// SIMATIC STEP 7 (V5.x) project R706_Cogeme_V_0_2
// CPU: CPU 315-2 DP
// station: Hardware
// station: R706_Ass_3PCS_Insert
// station: P_ADR_BUS
// program: Programma S7(1)
// program: Backup  DB 20100406
// program: SINAMICS_S120_CU310_DP
// program: SINAMICS_S120_CU310_DP

SYMBOL_TABLE
"Line"	DB 50	UDT 250
"Line.MapE"	DB 51	DB 51
"Line.MapA"	DB 52	DB 52
"Line.Config"	DB 53	DB 53
"Line.Alarms"	DB 54	DB 54
"Line.Systems"	DB 55	DB 55
"Line.Cycles"	DB 60	DB 60
"Line.OperatorPanel"	DB 70	DB 70
"OP10"	DB 100	UDT 250
"Op10.Bench.MapE"	DB 101	DB 101
"Op10.Bench.MapA"	DB 102	DB 102
"Op10.Bench.Config"	DB 103	DB 103
"Op10.Bench.Alarms"	DB 104	DB 104
"Op10.Bench.Systems"	DB 105	DB 105
"Op10.Tools.MapE"	DB 106	DB 106
"Op10.Tools.Config"	DB 108	DB 108
"Op10.Tools.Systems"	DB 109	DB 109
"Op10.Bench.Recipe"	DB 110	DB 110
"Op10.Cycles"	DB 120	DB 120
"OP20"	DB 150	UDT 250
"Op20.Bench.MapE"	DB 151	DB 151
"Op20.Bench.MapA"	DB 152	DB 152
"Op20.Bench.Config"	DB 153	DB 153
"Op20.Bench.Alarms"	DB 154	DB 154
"Op20.Bench.Systems"	DB 155	DB 155
"Op20.Tools.MapE"	DB 156	DB 156
"Op20.Tools.Config"	DB 158	DB 158
"Op20.Tools.Systems"	DB 159	DB 159
"Op20.Bench.Recipe"	DB 160	DB 160
"Op20.Cycles"	DB 170	DB 170
"OP40"	DB 200	UDT 250
"Op40.Bench.MapE"	DB 201	DB 201
"Op40.Bench.MapA"	DB 202	DB 202
"Op40.Bench.Config"	DB 203	DB 203
"Op40.Bench.Alarms"	DB 204	DB 204
"Op40.Bench.Systems"	DB 205	DB 205
"Op40.Tools.MapE"	DB 206	DB 206
"Op40.Tools.Config"	DB 208	DB 208
"Op40.Tools.Systems"	DB 209	DB 209
"Op40.Bench.Recipe"	DB 210	DB 210
"Op40.Cycles"	DB 220	DB 220
"Op05.Bench"	DB 300	UDT 250
"Ist_cil_10_Index_cass"	DB 401	FB 102
"Ist_10_CilBloccoPezzo"	DB 402	FB 102
"Ist_cil_20_Index_cass"	DB 403	FB 102
"Ist_cil_20_gr_piantaggio"	DB 404	FB 102
"Ist_cil_20_piantaggio"	DB 405	FB 102
"Ist_cil_40_Index_cass"	DB 406	FB 102
"Ist_40_CilBloccoPezzo"	DB 407	FB 102
"Ist_AsseX"	DB 420	FB 450
"Ist_AsseY"	DB 421	FB 450
"Ist_CU_asseX"	DB 425	FB 455
"Ist_CU_asseY"	DB 426	FB 455
"Op10.Ist.Cycle.General"	DB 430	FB 120
"Op10.Ist.Cycle.Restore"	DB 431	FB 121
"OP40.Ist.Cycle.Restore"	DB 435	FB 221
"OP40.Ist.Cycle.General"	DB 436	FB 220
"OP20.Ist.Cycle.Restore"	DB 437	FB 171
"OP20.Ist.Cycle.General"	DB 438	FB 170
"Line.Ist.Cycle.Coord_rib"	DB 440	FB 60
"Line.Cycle.Coord_ribadit"	FB 60	FB 60	// Coordinamento ribaditrice
"Std System.Cylinder"	FB 102	FB 102
"Op10.Cycle.General"	FB 120	FB 120
"Op10.Cycle.Restore"	FB 121	FB 121
"Op20.Cycle.General"	FB 170	FB 170
"Op20.Cycle.Restore"	FB 171	FB 171
"Op40.Cycle.General"	FB 220	FB 220
"Op40.Cycle.Restore"	FB 221	FB 221
"Std_Sinamics_Axis"	FB 450	FB 450
"Std.Sinamics_Cu_S"	FB 455	FB 455
"SCALE"	FC 5	FC 5	// Scaling Values
"Conv_INT->BIT"	FC 17	FC 17
"Bench.Mode"	FC 20	FC 20
"Bench.Alarms"	FC 21	FC 21	// Da ricontrollare!!!!
"TIM_S5TI"	FC 40	FC 40	// IEC Time to S5 Time
"Line.FCMain"	FC 50	FC 50
"Line.FCMapE"	FC 51	FC 51
"Line.FCMapA"	FC 52	FC 52
"Line.FCConfig"	FC 53	FC 53
"Line.FCSystems"	FC 55	FC 55
"Line.FCCycles"	FC 60	FC 60
"Line.FCOperatorPanel"	FC 70	FC 70
"OP10.FCMain"	FC 100	FC 100
"Op10.Bench.FCMapE"	FC 101	FC 101
"Op10.Bench.FCMapA"	FC 102	FC 102
"Op10.Bench.FCConfig"	FC 103	FC 103
"Op10.Bench.FCSystems"	FC 105	FC 105
"Op10.Tool.FCMap.E"	FC 106	FC 106
"Op10.FCCycles"	FC 120	FC 120
"OP20.FCMain"	FC 150	FC 150
"Op20.Bench.FCMapE"	FC 151	FC 151
"Op20.Bench.FCMapA"	FC 152	FC 152
"Op20.Bench.FCConfig"	FC 153	FC 153
"Op20.Bench.FCSystems"	FC 155	FC 155
"Op20.Tool.FCMapE"	FC 156	FC 156
"Op20.FCCycles"	FC 170	FC 170
"OP40.FCMain"	FC 200	FC 200
"Op40.Bench.FCMapE"	FC 201	FC 201
"Op40.Bench.FCMapA"	FC 202	FC 202
"Op40.Bench.FCConfig"	FC 203	FC 203
"Op40.Bench.FCSystems"	FC 205	FC 205
"Op40.Tool.FCMapE"	FC 206	FC 206
"Op40.FCCycles"	FC 220	FC 220
"Dummy_ReferenceAxX"	M 10.0	BOOL
"Dummy_RefCamAxX"	M 10.1	BOOL
"Dummy_ReferenceAxY"	M 10.2	BOOL
"Dummy_RefCamAxY"	M 10.3	BOOL
"AppoFP_M50.0"	M 50.0	BOOL
"AppoFP_M50.1"	M 50.1	BOOL
"AppoFP_M50.2"	M 50.2	BOOL
"AppoFP_M50.3"	M 50.3	BOOL
"AppoFP_M50.4"	M 50.4	BOOL
"AppoFP_M50.5"	M 50.5	BOOL
"AppoFP_M50.6"	M 50.6	BOOL
"AppoFP_M50.7"	M 50.7	BOOL
"AppoFP_M51.0"	M 51.0	BOOL
"AppoFP_M51.1"	M 51.1	BOOL
"AppoFPM51.2"	M 51.2	BOOL
"AppoFPM51.3"	M 51.3	BOOL
"AppoFPM51.4"	M 51.4	BOOL
"AppoFPM51.5"	M 51.5	BOOL
"AppoFP_M51.6"	M 51.6	BOOL
"AppoFP_M51.7"	M 51.7	BOOL
"AppoFP_M52.0"	M 52.0	BOOL
"Alw_ON"	M 100.0	BOOL
"alw_OFF"	M 100.1	BOOL
"FirstScan"	M 100.2	BOOL
"M100.3"	M 100.3	BOOL
"FP_manual"	M 100.4	BOOL
"M100.5"	M 100.5	BOOL
"Fp_Automatic"	M 100.6	BOOL
"Clock-T=0,1 sec."	M 250.0	BOOL
"Clock-T=0,2 sec."	M 250.1	BOOL
"Clock-T=0,4 sec."	M 250.2	BOOL
"Clock-T=0,5 sec."	M 250.3	BOOL
"Clock-T=0,8 sec."	M 250.4	BOOL
"Clock-T=1 sec."	M 250.5	BOOL
"Clock-T=1,6 sec."	M 250.6	BOOL
"Clock-T=2 sec."	M 250.7	BOOL
"I/O_FLT1"	OB 82	OB 82	// I/O Point Fault 1
"RACK_FLT"	OB 86	OB 86	// Loss of Rack Fault
"TON"	SFB 4	SFB 4	// Generate an On Delay
"DPRD_DAT"	SFC 14	SFC 14	// Read Consistent Data of a Standard DP Slave
"DPWR_DAT"	SFC 15	SFC 15	// Write Consistent Data to a Standard DP Slave
"TempoResetAllarmi"	T 2	TIMER
"T_All_Rientro_PLC_OK"	T 3	TIMER
"T_Allarme_aria_compressa"	T 5	TIMER
"Rit_all_potre_non_blocc"	T 6	TIMER
"Op10_Tempo_di_ribaditura"	T 10	TIMER
"Op40_Tempo_di_ribaditura"	T 11	TIMER
"TOP20_Cassetto dentro"	T 20	TIMER
"OP20_TimeoutPiantaggio"	T 21	TIMER
"OP20_TempoDiPiantaggio"	T 22	TIMER
"OP10St13_Cassetto_dentro"	T 25	TIMER
"OP10St35_Cassetto_fuori"	T 26	TIMER
"RP10St15_Cassetto_fuori"	T 27	TIMER
"OP20ST10_Cassetto_dentro"	T 28	TIMER
"OP40St13_Cassetto_dentro"	T 29	TIMER
"OP40St35_Cassetto_fuori"	T 30	TIMER
"RS40St15_Cassetto_fuori"	T 31	TIMER
"Cycles_UDT"	UDT 200	UDT 200
"Bench_UDT"	UDT 250	UDT 250
"Sinamics Telegramma Assi"	UDT 450	UDT 450
"Sinamics TelegrammaCU_S"	UDT 455	UDT 455
"Assi e posizioni"	VAT 1	
END_SYMBOL_TABLE

TYPE "Cycles_UDT"	// UDT 200
VERSION : 0.1
  STRUCT
   State : STRUCT
    State : INT ;	//Stato del ciclo
    Page : INT ;	//Pagina
    Message : INT ;	//Messaggio
    Cycle_In_Progress : BOOL ;	//Ciclo in corso
    Cycle_Ended_OK : BOOL ;	//Ciclo terminato OK
    Cycle_Ended_KO : BOOL ;	//Ciclo terminato KO
    State_Bit : ARRAY  [0 .. 63 ] OF //Bit Stato
    BOOL ;
    Free : INT ;
   END_STRUCT ;
   Command : STRUCT
    Activate_Cycle : BOOL ;	//Attiva ciclo
    Hold_Cycle : BOOL ;	//Sospendi ciclo
    Single_Step : BOOL ;	//Passo singolo
    Lock_Outputs : BOOL ;	//Blocco uscite
    Free : INT ;
   END_STRUCT ;
  END_STRUCT ;	
END_TYPE

TYPE "Bench_UDT"	// UDT 250
VERSION : 0.1
  STRUCT
   Mode : STRUCT
    Emergency : BOOL ;	//MODO Macchina spenta
    Test_Machine : BOOL ;	//MODO Aspetta pressione nel circuito pneumatico e/o idraulico + MODO Test Lampad
    Setup : BOOL ;	//MODO Cambio Ricetta o setup
    Manual : BOOL ;	//MODO Manuale
    Automatic : BOOL ;	//MODO Automatico
    Service : BOOL ;	//MODO Messa in servizio
    Free_06 : BOOL ;
    Free_07 : BOOL ;
   END_STRUCT ;
   Diagnostic : STRUCT
    Alarm_Emergency : BOOL ;	//Macchina in Emergenza
    Alarm_Stop_Cycle : BOOL ;	//Allarme che blocca il ciclo attivo
    Alarm_No_Restart : BOOL ;	//Allarme che blocca un nuovo ciclo
    Alarm_Warning : BOOL ;	//Segnalazione o avvertenza
    Safe_State : BOOL ;	//MODO Sicuro : e' possibile eseguire i comandi manuali in sicurezza
    Initial_Conditions : BOOL ;	//condizioni iniziali macchina
    Hold_State : BOOL ;	//Hold Macchina
    Free_07 : BOOL ;
    ResetAlarm : BOOL ;
   END_STRUCT ;
   Software : STRUCT
    SwName : STRING  [20 ];
    SwVersion : STRING  [11 ];
   END_STRUCT ;
  END_STRUCT ;	
END_TYPE

TYPE "Sinamics Telegramma Assi"	// UDT 450
AUTHOR : Castel
VERSION : 0.1
  STRUCT
   IN : STRUCT
    IN_PZD1_BIT8 : BOOL ;	//PAST1 Bit8 distanza di inseguimento nella tolleranza (1=si 0=no)
    IN_PZD1_BIT9 : BOOL ;	//PAST1 Bit9 comando richiesto (1=si 0=no)
    IN_PZD1_BIT10 : BOOL ;	//PAST1 Bit10 posizione di destinazione raggiunta (1=si 0=no)
    IN_PZD1_BIT11 : BOOL ;	//PAST1 Bit11 punto di riferimento impostato (1=si 0=no)
    IN_PZD1_BIT12 : BOOL ;	//PAST1 Bit12 tacitazione blocco movimento attivata (1=si 0=no)
    IN_PZD1_BIT13 : BOOL ;	//PAST1 Bit13 (motore fermo) n_att< valore di soglia num.giri 3 P2161 (1=si 0=no)
    IN_PZD1_BIT14 : BOOL ;	//PAST1 Bit14 riservato
    IN_PZD1_BIT15 : BOOL ;	//PAST1 Bit15 riservato
    IN_PZD1_BIT0 : BOOL ;	//PAST1 Bit0 pronto all'inserzione (1=si 0=no)
    IN_PZD1_BIT1 : BOOL ;	//PAST1 Bit1 pronto al funzionamento (1=si 0=no)
    IN_PZD1_BIT2 : BOOL ;	//PAST1 Bit2 funzionamento abilitazione (1=si 0=no)
    IN_PZD1_BIT3 : BOOL ;	//PAST1 Bit3 anomalia attiva (1=si 0=no)
    IN_PZD1_BIT4 : BOOL ;	//PAST1 Bit4 nessun arresto per inerzia attivo (1=OFF2 inattivo 0=OFF2 attivo)
    IN_PZD1_BIT5 : BOOL ;	//PAST1 Bit5 nessun arresto rapido attivo (1=OFF3 inattivo 0=OFF3 attivo)
    IN_PZD1_BIT6 : BOOL ;	//PAST1 Bit6 blocco inserzione attivo (1=si 0=no)
    IN_PZD1_BIT7 : BOOL ;	//PAST1 Bit7 avviso attivo (1=si 0=no)
    IN_PZD2_BIT8 : BOOL ;	//AKTSATZ Bit8
    IN_PZD2_BIT9 : BOOL ;	//AKTSATZ Bit9
    IN_PZD2_BIT10 : BOOL ;	//AKTSATZ Bit10
    IN_PZD2_BIT11 : BOOL ;	//AKTSATZ Bit11
    IN_PZD2_BIT12 : BOOL ;	//AKTSATZ Bit12
    IN_PZD2_BIT13 : BOOL ;	//AKTSATZ Bit13
    IN_PZD2_BIT14 : BOOL ;	//AKTSATZ Bit14 attivare il cambio del blocco esterno
    IN_PZD2_BIT15 : BOOL ;	//AKTSATZ Bit15 MDI attivo (1=attivo 0=inattivo)
    IN_PZD2_BIT0 : BOOL ;	//AKTSATZ Bit0 blocco di movimento attivo valenza 0 (1=attivo 0=inattivo)
    IN_PZD2_BIT1 : BOOL ;	//AKTSATZ Bit1 blocco di movimento attivo valenza 2 (1=attivo 0=inattivo)
    IN_PZD2_BIT2 : BOOL ;	//AKTSATZ Bit2 blocco di movimento attivo valenza 4 (1=attivo 0=inattivo)
    IN_PZD2_BIT3 : BOOL ;	//AKTSATZ Bit3 blocco di movimento attivo valenza 8 (1=attivo 0=inattivo)
    IN_PZD2_BIT4 : BOOL ;	//AKTSATZ Bit4 blocco di movimento attivo valenza 16 (1=attivo 0=inattivo)
    IN_PZD2_BIT5 : BOOL ;	//AKTSATZ Bit5 blocco di movimento attivo valenza 32 (1=attivo 0=inattivo)
    IN_PZD2_BIT6 : BOOL ;	//AKTSATZ Bit6
    IN_PZD2_BIT7 : BOOL ;	//AKTSATZ Bit7
    IN_PZD3_BIT8 : BOOL ;	//POSPAST Bit8 valore attuale di posiz. <= posiz.commutazione camma 1 (1=si 0=no)
    IN_PZD3_BIT9 : BOOL ;	//POSPAST Bit9 valore attuale di posiz. <= posiz.commutazione camma 2 (1=si 0=no)
    IN_PZD3_BIT10 : BOOL ;	//POSPAST Bit10 uscita diretta 1 su blocco di movimento (1=si 0=no)
    IN_PZD3_BIT11 : BOOL ;	//POSPAST Bit11 uscita diretta 2 su blocco di movimento (1=si 0=no)
    IN_PZD3_BIT12 : BOOL ;	//POSPAST Bit12
    IN_PZD3_BIT13 : BOOL ;	//POSPAST Bit13
    IN_PZD3_BIT14 : BOOL ;	//POSPAST Bit14
    IN_PZD3_BIT15 : BOOL ;	//POSPAST Bit15
    IN_PZD3_BIT0 : BOOL ;	//POSPAST Bit0 funzionamento a seguire attivo (1=si 0=no)
    IN_PZD3_BIT1 : BOOL ;	//POSPAST Bit1 limitazione di velocità attiva (1=si 0=no)
    IN_PZD3_BIT2 : BOOL ;	//POSPAST Bit2 valore di riferimento fermo (1=si 0=no)
    IN_PZD3_BIT3 : BOOL ;	//POSPAST Bit3
    IN_PZD3_BIT4 : BOOL ;	//POSPAST Bit4 asse in movimento avanti (1=si 0=no)
    IN_PZD3_BIT5 : BOOL ;	//POSPAST Bit5 asse in movimento indietro (1=si 0=no)
    IN_PZD3_BIT6 : BOOL ;	//POSPAST Bit6 finecorsa software meno raggiunto (1=si 0=no)
    IN_PZD3_BIT7 : BOOL ;	//POSPAST Bit7 finecorsa software più raggiunto (1=si 0=no)
    IN_PZD4_BIT8 : BOOL ;	//PAST2 Bit8 posizionamento su riscontro fisso attivo (1=si 0=no)
    IN_PZD4_BIT9 : BOOL ;	//PAST2 Bit9
    IN_PZD4_BIT10 : BOOL ;	//PAST2 Bit10
    IN_PZD4_BIT11 : BOOL ;	//PAST2 Bit11 commutazione record di dati motore attiva (1=attivo 0=inattivo)
    IN_PZD4_BIT12 : BOOL ;	//PAST2 Bit12 segno di vita dello slave bit 0 (1=on 0=off)
    IN_PZD4_BIT13 : BOOL ;	//PAST2 Bit13 segno di vita dello slave bit 1 (1=on 0=off)
    IN_PZD4_BIT14 : BOOL ;	//PAST2 Bit14 segno di vita dello slave bit 2 (1=on 0=off)
    IN_PZD4_BIT15 : BOOL ;	//PAST2 Bit15 segno di vita dello slave bit 3 (1=on 0=off)
    IN_PZD4_BIT0 : BOOL ;	//PAST2 Bit0 DDS attivo bit 0 (1=on 0=off)
    IN_PZD4_BIT1 : BOOL ;	//PAST2 Bit1 DDS attivo bit 1 (1=on 0=off)
    IN_PZD4_BIT2 : BOOL ;	//PAST2 Bit2 DDS attivo bit 2 (1=on 0=off)
    IN_PZD4_BIT3 : BOOL ;	//PAST2 Bit3 DDS attivo bit 3 (1=on 0=off)
    IN_PZD4_BIT4 : BOOL ;	//PAST2 Bit4 DDS attivo bit 4 (1=on 0=off)
    IN_PZD4_BIT5 : BOOL ;	//PAST2 Bit5
    IN_PZD4_BIT6 : BOOL ;	//PAST2 Bit6
    IN_PZD4_BIT7 : BOOL ;	//PAST2 Bit7 asse in sosta attivo (1=si 0=no)
    IN_PZD5_BIT8 : BOOL ;	//SEGNW Bit8 diff.val.rif./att.n.giri entro tolleranza t_on (1=si 0=no)
    IN_PZD5_BIT9 : BOOL ;	//SEGNW Bit9
    IN_PZD5_BIT10 : BOOL ;	//SEGNW Bit10
    IN_PZD5_BIT11 : BOOL ;	//SEGNW Bit11 abilitazione regolatore (1=si 0=no)
    IN_PZD5_BIT12 : BOOL ;	//SEGNW Bit12 azionamento pronto (1=si 0=no)
    IN_PZD5_BIT13 : BOOL ;	//SEGNW Bit13 impulsi abilitati (1=si 0=no)
    IN_PZD5_BIT14 : BOOL ;	//SEGNW Bit14
    IN_PZD5_BIT15 : BOOL ;	//SEGNW Bit15
    IN_PZD5_BIT0 : BOOL ;	//SEGNW Bit0 accelerazione/decelerazione conclusa (1=si 0=no)
    IN_PZD5_BIT1 : BOOL ;	//SEGNW Bit1 utilizzo della coppia< soglia di coppia 2 (1=si 0=no)
    IN_PZD5_BIT2 : BOOL ;	//SEGNW Bit2 n_att<valore di soglia numero di giri 3 (1=si 0=no)
    IN_PZD5_BIT3 : BOOL ;	//SEGNW Bit3 n_att<valore di soglia numero di giri 2 (1=si 0=no)
    IN_PZD5_BIT4 : BOOL ;	//SEGNW Bit4
    IN_PZD5_BIT5 : BOOL ;	//SEGNW Bit5
    IN_PZD5_BIT6 : BOOL ;	//SEGNW Bit6 avviso surriscaldamento motore (1=no 0=si)
    IN_PZD5_BIT7 : BOOL ;	//SEGNW Bit7 avviso sovraccarico termico modulo di potenza (1=no 0=si)
    IN_PZD6_7 : DINT ;	//XISTP posizione attuale asse in micron
   END_STRUCT ;
   OUT : STRUCT
    OUT_PZD1_BIT8 : BOOL ;	//PACO1 Bit8 EPOS funzionamento a impulsi jog negativo
    OUT_PZD1_BIT9 : BOOL ;	//PACO1 Bit9 EPOS funzionamento a impulsi jog positivo
    OUT_PZD1_BIT10 : BOOL ;	//PACO1 Bit10 controllo da plc (abilitazione profibus)
    OUT_PZD1_BIT11 : BOOL ;	//PACO1 Bit11 EPOS avvio ricerca punto di riferimento
    OUT_PZD1_BIT12 : BOOL ;	//PACO1 Bit12
    OUT_PZD1_BIT13 : BOOL ;	//PACO1 Bit13
    OUT_PZD1_BIT14 : BOOL ;	//PACO1 Bit14
    OUT_PZD1_BIT15 : BOOL ;	//PACO1 Bit15
    OUT_PZD1_BIT0 : BOOL ;	//PACO1 Bit0 0=OFF1 arresto tramite datore di rampa
    OUT_PZD1_BIT1 : BOOL ;	//PACO1 Bit1 0=OFF2 blocco impulsi
    OUT_PZD1_BIT2 : BOOL ;	//PACO1 Bit2 0=OFF3 arresto rapido
    OUT_PZD1_BIT3 : BOOL ;	//PACO1 Bit3 abilitazione funzionamento
    OUT_PZD1_BIT4 : BOOL ;	//PACO1 Bit4 EPOS rifuito job di movimento (segnale 0)
    OUT_PZD1_BIT5 : BOOL ;	//PACO1 Bit5 EPOS arresto intermedio (segnale 0)
    OUT_PZD1_BIT6 : BOOL ;	//PACO1 Bit6 EPOS attivazione job di movimento (impulso 0->1)
    OUT_PZD1_BIT7 : BOOL ;	//PACO1 Bit7 tacitazione anomalie
    OUT_PZD2_BIT8 : BOOL ;	//SCELBLOC Bit8
    OUT_PZD2_BIT9 : BOOL ;	//SCELBLOC Bit9
    OUT_PZD2_BIT10 : BOOL ;	//SCELBLOC Bit10
    OUT_PZD2_BIT11 : BOOL ;	//SCELBLOC Bit11
    OUT_PZD2_BIT12 : BOOL ;	//SCELBLOC Bit12
    OUT_PZD2_BIT13 : BOOL ;	//SCELBLOC Bit13
    OUT_PZD2_BIT14 : BOOL ;	//SCELBLOC Bit14
    OUT_PZD2_BIT15 : BOOL ;	//SCELBLOC Bit15 EPOS impostazione diretta val.di riferimento/attivare MDI
    OUT_PZD2_BIT0 : BOOL ;	//SCELBLOC Bit0 EPOS selezione blocco valenza 1
    OUT_PZD2_BIT1 : BOOL ;	//SCELBLOC Bit1 EPOS selezione blocco valenza 2
    OUT_PZD2_BIT2 : BOOL ;	//SCELBLOC Bit2 EPOS selezione blocco valenza 4
    OUT_PZD2_BIT3 : BOOL ;	//SCELBLOC Bit3 EPOS selezione blocco valenza 8
    OUT_PZD2_BIT4 : BOOL ;	//SCELBLOC Bit4 EPOS selezione blocco valenza 16
    OUT_PZD2_BIT5 : BOOL ;	//SCELBLOC Bit5 EPOS selezione blocco valenza 32
    OUT_PZD2_BIT6 : BOOL ;	//SCELBLOC Bit6
    OUT_PZD2_BIT7 : BOOL ;	//SCELBLOC Bit7
    OUT_PZD3_BIT8 : BOOL ;	//POSPACO Bit8
    OUT_PZD3_BIT9 : BOOL ;	//POSPACO Bit9
    OUT_PZD3_BIT10 : BOOL ;	//POSPACO Bit10
    OUT_PZD3_BIT11 : BOOL ;	//POSPACO Bit11
    OUT_PZD3_BIT12 : BOOL ;	//POSPACO Bit12
    OUT_PZD3_BIT13 : BOOL ;	//POSPACO Bit13
    OUT_PZD3_BIT14 : BOOL ;	//POSPACO Bit14
    OUT_PZD3_BIT15 : BOOL ;	//POSPACO Bit15
    OUT_PZD3_BIT0 : BOOL ;	//POSPACO Bit0 EPOS selezione funzionamento a seguire
    OUT_PZD3_BIT1 : BOOL ;	//POSPACO Bit1 EPOS impostazione punto riferimento
    OUT_PZD3_BIT2 : BOOL ;	//POSPACO Bit2 EPOS ricerca punto di riferimento, camma di riferimento
    OUT_PZD3_BIT3 : BOOL ;	//POSPACO Bit3
    OUT_PZD3_BIT4 : BOOL ;	//POSPACO Bit4
    OUT_PZD3_BIT5 : BOOL ;	//POSPACO Bit5 EPOS funzionamento a impulsi incrementale
    OUT_PZD3_BIT6 : BOOL ;	//POSPACO Bit6
    OUT_PZD3_BIT7 : BOOL ;	//POSPACO Bit7
    OUT_PZD4_BIT8 : BOOL ;	//PACO2 Bit8 avanzamento su riscontro fisso, attivazione
    OUT_PZD4_BIT9 : BOOL ;	//PACO2 Bit9
    OUT_PZD4_BIT10 : BOOL ;	//PACO2 Bit10
    OUT_PZD4_BIT11 : BOOL ;	//PACO2 Bit11 commutazione motore, risposta di conferma
    OUT_PZD4_BIT12 : BOOL ;	//PACO2 Bit12 segno di vita bit 0
    OUT_PZD4_BIT13 : BOOL ;	//PACO2 Bit13 segno di vita bit 1
    OUT_PZD4_BIT14 : BOOL ;	//PACO2 Bit14 segno di vita bit 3
    OUT_PZD4_BIT15 : BOOL ;	//PACO2 Bit15 segno di vita bit 4
    OUT_PZD4_BIT0 : BOOL ;	//PACO2 Bit0 selezione record di dati azionamento DDS bit 0
    OUT_PZD4_BIT1 : BOOL ;	//PACO2 Bit1 selezione record di dati azionamento DDS bit 1
    OUT_PZD4_BIT2 : BOOL ;	//PACO2 Bit2 selezione record di dati azionamento DDS bit 2
    OUT_PZD4_BIT3 : BOOL ;	//PACO2 Bit3 selezione record di dati azionamento DDS bit 3
    OUT_PZD4_BIT4 : BOOL ;	//PACO2 Bit4 selezione record di dati azionamento DDS bit 4
    OUT_PZD4_BIT5 : BOOL ;	//PACO2 Bit5
    OUT_PZD4_BIT6 : BOOL ;	//PACO2 Bit6
    OUT_PZD4_BIT7 : BOOL ;	//PACO2 Bit7 selezione asse in sosta
    OUT_PZD5 : INT ;	//OVER override asse 0..32767
    OUT_PZD6_7 : DINT ;	//MDIPOS posizione in micron
    OUT_PZD8_9 : DINT ;	//MDIVEL velocità lineare asse 0..30000
    OUT_PZD10 : INT ;	//MDIACC accelerazione 0..32767
    OUT_PZD11 : INT ;	//MDIDEC decelerazione 0..32767
    OUT_PZD12 : INT ;	//MDIMODE
   END_STRUCT ;
  END_STRUCT ;	
END_TYPE

TYPE "Sinamics TelegrammaCU_S"	// UDT 455
AUTHOR : Castel
VERSION : 0.1
  STRUCT
   IN : STRUCT
    IN_PZD1_BIT8 : BOOL ;	//PAST1 Bit8 ora di sistema sincronizzata (1=si 0=no)
    IN_PZD1_BIT9 : BOOL ;	//PAST1 Bit9
    IN_PZD1_BIT10 : BOOL ;	//PAST1 Bit10
    IN_PZD1_BIT11 : BOOL ;	//PAST1 Bit11
    IN_PZD1_BIT12 : BOOL ;	//PAST1 Bit12 funzionalita vitale slave bit0 (1=si 0=no)
    IN_PZD1_BIT13 : BOOL ;	//PAST1 Bit13 funzionalita vitale slave bit1 (1=si 0=no)
    IN_PZD1_BIT14 : BOOL ;	//PAST1 Bit14 funzionalita vitale slave bit2 (1=si 0=no)
    IN_PZD1_BIT15 : BOOL ;	//PAST1 Bit15 funzionalita vitale slave bit3 (1=si 0=no)
    IN_PZD1_BIT0 : BOOL ;	//PAST1 Bit0
    IN_PZD1_BIT1 : BOOL ;	//PAST1 Bit1
    IN_PZD1_BIT2 : BOOL ;	//PAST1 Bit2
    IN_PZD1_BIT3 : BOOL ;	//PAST1 Bit3 anomalia attiva (1=si 0=no)
    IN_PZD1_BIT4 : BOOL ;	//PAST1 Bit4
    IN_PZD1_BIT5 : BOOL ;	//PAST1 Bit5
    IN_PZD1_BIT6 : BOOL ;	//PAST1 Bit6
    IN_PZD1_BIT7 : BOOL ;	//PAST1 Bit7 avviso attivo (1=si 0=no)
    IN_PZD2_BIT8 : BOOL ;	//E_DIGITAL Bit8 CU mors.DI 0 (X122.1/X121.1) [Reset allarmi]
    IN_PZD2_BIT9 : BOOL ;	//E_DIGITAL Bit9 CU mors.DI 1 (X122.2/X121.2) [Emergenza istantanea]
    IN_PZD2_BIT10 : BOOL ;	//E_DIGITAL Bit10 CU mors.DI 2 (X122.3/X121.3) [Emergenza ritardata]
    IN_PZD2_BIT11 : BOOL ;	//E_DIGITAL Bit11 CU mors.DI 3 (X122.4/X121.4) [Alimentatore OK]
    IN_PZD2_BIT12 : BOOL ;	//E_DIGITAL Bit12 CU mors.DI 4 (X132.1) [Finecorsa Harware asse Y+]
    IN_PZD2_BIT13 : BOOL ;	//E_DIGITAL Bit13 CU mors.DI 5 (X132.2) [Finecorsa Harware asse Y-]
    IN_PZD2_BIT14 : BOOL ;	//E_DIGITAL Bit14 CU mors.DI 6 (X132.3) [Finecorsa Harware asse X+]
    IN_PZD2_BIT15 : BOOL ;	//E_DIGITAL Bit15 CU mors.DI 7 (X132.4) [Finecorsa Harware asse X-]
    IN_PZD2_BIT0 : BOOL ;	//E_DIGITAL Bit0 CU mors.DI 8 (X122.7/X121.7)
    IN_PZD2_BIT1 : BOOL ;	//E_DIGITAL Bit1 CU mors.DI 9 (X122.8/X121.8)
    IN_PZD2_BIT2 : BOOL ;	//E_DIGITAL Bit2 CU mors.DI 10 (X122.10/X121.10)
    IN_PZD2_BIT3 : BOOL ;	//E_DIGITAL Bit3 CU mors.DI 11 (X122.11/X121.11)
    IN_PZD2_BIT4 : BOOL ;	//E_DIGITAL Bit4 CU mors.DI 12 (X132.7) [Finecorsa Harware asse Z+]
    IN_PZD2_BIT5 : BOOL ;	//E_DIGITAL Bit5 CU mors.DI 13 (X132.8) [Finecorsa Harware asse Z-]
    IN_PZD2_BIT6 : BOOL ;	//E_DIGITAL Bit6 CU mors.DI 14 (X132.10)
    IN_PZD2_BIT7 : BOOL ;	//E_DIGITAL Bit7 CU mors.DI 15 (X132.11)
   END_STRUCT ;
   OUT : STRUCT
    OUT_PZD1_BIT8 : BOOL ;	//PACO1 Bit8
    OUT_PZD1_BIT9 : BOOL ;	//PACO1 Bit9
    OUT_PZD1_BIT10 : BOOL ;	//PACO1 Bit10
    OUT_PZD1_BIT11 : BOOL ;	//PACO1 Bit11
    OUT_PZD1_BIT12 : BOOL ;	//PACO1 Bit12
    OUT_PZD1_BIT13 : BOOL ;	//PACO1 Bit13
    OUT_PZD1_BIT14 : BOOL ;	//PACO1 Bit14
    OUT_PZD1_BIT15 : BOOL ;	//PACO1 Bit15
    OUT_PZD1_BIT0 : BOOL ;	//PACO1 Bit0 sorgente del segnale di sincronizzazione tastatore centrale
    OUT_PZD1_BIT1 : BOOL ;	//PACO1 Bit1 RTC sincronizzazione in tempo reale PING
    OUT_PZD1_BIT2 : BOOL ;	//PACO1 Bit2
    OUT_PZD1_BIT3 : BOOL ;	//PACO1 Bit3
    OUT_PZD1_BIT4 : BOOL ;	//PACO1 Bit4
    OUT_PZD1_BIT5 : BOOL ;	//PACO1 Bit5
    OUT_PZD1_BIT6 : BOOL ;	//PACO1 Bit6
    OUT_PZD1_BIT7 : BOOL ;	//PACO1 Bit7 tacitazione anomalie
    OUT_PZD2_BIT8 : BOOL ;	//A_DIGITAL Bit8
    OUT_PZD2_BIT9 : BOOL ;	//A_DIGITAL Bit9
    OUT_PZD2_BIT10 : BOOL ;	//A_DIGITAL Bit10
    OUT_PZD2_BIT11 : BOOL ;	//A_DIGITAL Bit11
    OUT_PZD2_BIT12 : BOOL ;	//A_DIGITAL Bit12
    OUT_PZD2_BIT13 : BOOL ;	//A_DIGITAL Bit13
    OUT_PZD2_BIT14 : BOOL ;	//A_DIGITAL Bit14
    OUT_PZD2_BIT15 : BOOL ;	//A_DIGITAL Bit15
    OUT_PZD2_BIT0 : BOOL ;	//A_DIGITAL Bit0 CU mors.DI/DO 8 (X122.7/X121.7) [Sinamics in fault]
    OUT_PZD2_BIT1 : BOOL ;	//A_DIGITAL Bit1 CU mors.DI/DO 9 [Sinamics pronto]
    OUT_PZD2_BIT2 : BOOL ;	//A_DIGITAL Bit2 CU mors.DI/DO 10 [Assi fermi in sicurezza]
    OUT_PZD2_BIT3 : BOOL ;	//A_DIGITAL Bit3 CU mors.DI/DO 11
    OUT_PZD2_BIT4 : BOOL ;	//A_DIGITAL Bit4 CU mors.DI/DO 12
    OUT_PZD2_BIT5 : BOOL ;	//A_DIGITAL Bit5 CU mors.DI/DO 13
    OUT_PZD2_BIT6 : BOOL ;	//A_DIGITAL Bit6 CU mors.DI/DO 14
    OUT_PZD2_BIT7 : BOOL ;	//A_DIGITAL Bit7 CU mors.DI/DO 15
   END_STRUCT ;
  END_STRUCT ;	
END_TYPE

FUNCTION_BLOCK "Line.Cycle.Coord_ribadit"	// FB 60
VERSION : 0.1
VAR_INPUT
  IN_Cm_ON : BOOL ;	//1: Attiva il ciclo; 0: Reset del ciclo
  IN_HOLD : BOOL ;	//Blocca il ciclo nel passo successivo
  IN_STEP : BOOL ;
END_VAR
VAR_OUTPUT
  OUT_St_CicloInCorso : BOOL ;
  OUT_St_CicloTerminatoOK : BOOL ;
  OUT_St_CicloTerminatoKO : BOOL ;
  OUT_CicloStato : INT ;
  OUT_Page : INT ;
  OUT_Message : INT ;
END_VAR
VAR
  Stato : INT ;
  StatoSeguente : INT ;
  FrontePassoSingolo : BOOL ;
  Stat_CicloTermOk : BOOL ;
  Stat_CicloTermKO : BOOL ;
  Stat_CicloInCorso : BOOL ;
  Timer_Pennarello : SFB 4;
END_VAR
VAR_TEMP
  Pag_Active : ARRAY  [0 .. 100 ] OF BOOL ;
END_VAR
BEGIN
NETWORK
TITLE = FLOW CHART
NETWORK
TITLE = Update state
      A     #IN_Cm_ON;
      JC    M002;
      L     0;
      T     #Stato;
      T     #StatoSeguente;
M002: NOP   0;
//->Update State
      A     #IN_STEP;
      FP    #FrontePassoSingolo;
      ON    #IN_HOLD;	//se usassi UN l'Hold agirebbe anche su avanzamento a passo singolo 
      JCN   N100;
      L     #StatoSeguente;
      T     #Stato;
N100: NOP   0;
// determinazione bit di stato
      CALL  "Conv_INT->BIT" (
           Valore                   := #Stato,
           States                   := "Line.Cycles".Coord_Ribaditrice.State.State_Bit);
NETWORK
TITLE = Detect page active from OP
// serve??????
//      CALL  "Conv_INT->BIT"
//       Valore:=DB325.DBW2
//       States:=#Pag_Active
NETWORK
TITLE = States particular
      L     #Stato;
      L     0;
      <>I;
//->Evita ritardi
      A     #IN_Cm_ON;
      =     #Stat_CicloInCorso;
      A     "Line.Cycles".Coord_Ribaditrice.State.State_Bit[60];
      =     #Stat_CicloTermOk;
      A     "Line.Cycles".Coord_Ribaditrice.State.State_Bit[63];
      =     #Stat_CicloTermKO;
NETWORK
TITLE = Diagnostic default
//    L     0
//    T     #Page
//    L     0
//    T     #Message 
//      L     6
//      T     #StatoSeguente
NETWORK
TITLE = State <0>: Ciclo off
      A     "Line.Cycles".Coord_Ribaditrice.State.State_Bit[0];
      JCN   Z000;
      A     #IN_Cm_ON;
      A     "Line.Systems".Command.PrenotaRib_OP10;
      JC    Y000;
      A     #IN_Cm_ON;
      A     "Line.Systems".Command.PrenotaRib_OP40;
      JC    X000;
      JU    Z000;
Y000: L     10;
      T     #StatoSeguente;
      JU    Z000;
X000: L     20;
      T     #StatoSeguente;
Z000: NOP   0;
NETWORK
TITLE = State <10>: Ribaditrice prenotata da OP10
      A     "Line.Cycles".Coord_Ribaditrice.State.State_Bit[10];
      JCN   Z010;
      AN    "Line.Systems".Command.PrenotaRib_OP10;
      JC    Y010;
      JU    Z010;
// Stati di destinazione
Y010: L     0;
      T     #StatoSeguente;
Z010: NOP   0;
NETWORK
TITLE = State <20>: Ribaditrice prenotata da OP40
      A     "Line.Cycles".Coord_Ribaditrice.State.State_Bit[20];
      JCN   Z020;
      AN    "Line.Systems".Command.PrenotaRib_OP40;
      JC    Y020;
      JU    Z020;
// Stati di destinazione
Y020: L     0;
      T     #StatoSeguente;
Z020: NOP   0;
NETWORK
TITLE = Output
      L     #Stato;
      T     #OUT_CicloStato;
      A     #Stat_CicloInCorso;
      =     #OUT_St_CicloInCorso;
      A     #Stat_CicloTermOk;
      =     #OUT_St_CicloTerminatoOK;
      A     #Stat_CicloTermKO;
      =     #OUT_St_CicloTerminatoKO;
END_FUNCTION_BLOCK

FUNCTION_BLOCK "Std System.Cylinder"	// FB 102
VERSION : 2.1
VAR_INPUT
  IN_Enable : BOOL ;	//Abilita/Disabilita le uscite e gli allarmi
  IN_Command_CylForward : BOOL ;	//Se a 1 e non in hold comanda l'elettrovalvola
  IN_Command_CylBack : BOOL ;	//Se a 1 e non in hold comanda l'elettrovalvola
  IN_EndStroke_Forward : BOOL ;	//Ingresso PLC E...
  IN_EndStroke_Back : BOOL ;	//Ingresso PLC E...
  IN_Alarms_Reset : BOOL ;	//Tasto di reset allarme (fronte interno)
  IN_Alarms_TimeOut : TIME ;	//Tempo in secondi per time-out rilevamento Fc dopo comando
  IN_Hold_Condition : BOOL ;	//Condizione di hold cilindro durante movimento
END_VAR
VAR_OUTPUT
  OUT_EV_Forward : BOOL ;	//Uscita PLC A..
  OUT_EV_Back : BOOL ;	//Uscita PLC A..
  OUT_State_CylForward : BOOL ;	//Stato cilindro avanti
  OUT_State_CylBack : BOOL ;	//Stato cilindro indietro
  OUT_Alarm_ES_Forward : BOOL ;	//Allarme finecorsa avanti
  OUT_Alarm_ES_Back : BOOL ;	//Allarme finecorsa indietro
  OUT_Alarm_ForwBack : BOOL ;	//Allarme corto micro
  OUT_State_CylHold : BOOL ;	//Cilindro in stato di hold
END_VAR
VAR
  FP_IN_Comando_Avanti : BOOL ;
  FP_IN_Comando_Indietro : BOOL ;
  FP_ResetAllarmi : BOOL ;
  Timer1 : SFB 4;
  Timer2 : SFB 4;
END_VAR
VAR_TEMP
  Timer1_IN : BOOL ;
  Timer1_OUT : BOOL ;
  Timer2_IN : BOOL ;
  Timer2_OUT : BOOL ;
END_VAR
BEGIN
NETWORK
TITLE = FUNZIONE CILINDRO
//START CASE
// CASE: OFF
// CASE: ON
// CASE: DIS
//END CASE
//STATES
//HOLD
//ALARMS RESET
// ALLARM ON
// ALLARM OFF
// ALLARM ON OFF
NETWORK
TITLE =
      A     #IN_Alarms_Reset;
      A(;
      A     #IN_EndStroke_Forward;
      O     #IN_EndStroke_Back;
      );
      R     #OUT_State_CylHold;
NETWORK
TITLE = Select Case
//Condizioni per uscite elettrovalvole
      A     #IN_Command_CylForward;
      FP    #FP_IN_Comando_Avanti;
      O(;
      A     #IN_Command_CylBack;
      FP    #FP_IN_Comando_Indietro;
      );
      AN    #IN_Hold_Condition;
      R     #OUT_State_CylHold;
      AN    #IN_Enable;
      O     #OUT_State_CylHold;
      JC    DIS;
//-
      A     #IN_Command_CylForward;
      AN    #IN_Hold_Condition;
      JC    AV;
//-
      A     #IN_Command_CylBack;
      AN    #IN_Hold_Condition;
      JC    IND;
//-
      JU    ENDC;
NETWORK
TITLE = CASE: OFF
// Cilindro comandato in posizione "riposo"
IND:  NOP   0;
      SET;
      S     #OUT_EV_Back;
      R     #OUT_EV_Forward;
      JU    ENDC;
NETWORK
TITLE = CASE: ON
// Cilindro comandato in posizione "attivo"
AV:   NOP   0;
      SET;
      R     #OUT_EV_Back;
      S     #OUT_EV_Forward;
      JU    ENDC;
NETWORK
TITLE = CASE: DISABLE
// Uscite disabilitate
DIS:  NOP   0;
      SET;
      R     #OUT_EV_Back;
      R     #OUT_EV_Forward;
NETWORK
TITLE = END CASE
ENDC: NOP   0;
NETWORK
TITLE = STATES
// Cilindro in posizione "attivo"
      A     #IN_EndStroke_Forward;
      AN    #IN_EndStroke_Back;
      AN    #OUT_State_CylHold;
      =     #OUT_State_CylForward;
// Cilindro in posizione "riposo"
      AN    #IN_EndStroke_Forward;
      A     #IN_EndStroke_Back;
      AN    #OUT_State_CylHold;
      =     #OUT_State_CylBack;
NETWORK
TITLE = HOLD
// Abilita hold se barriera durante movimento
      A(;
      A     #OUT_EV_Forward;
      AN    #OUT_State_CylForward;
      A     #IN_Hold_Condition;
      O;
      A     #OUT_EV_Back;
      AN    #OUT_State_CylBack;
      A     #IN_Hold_Condition;
      );
      A     #IN_Enable;
      S     #OUT_State_CylHold;
NETWORK
TITLE = ALARMS RESET
// Reset allarmi
      A     #IN_Alarms_Reset;
      FP    #FP_ResetAllarmi;
      R     #OUT_Alarm_ES_Forward;
      R     #OUT_Alarm_ES_Back;
      R     #OUT_Alarm_ForwBack;
NETWORK
TITLE = Allarme Cilindro avanti non segnalato
// Cilindro non spostato in posizione "attivo" in tempo utile
      A     #OUT_EV_Forward;
      AN    #OUT_State_CylForward;
      AN    #IN_Hold_Condition;
      A     #IN_Enable;
      =     #Timer1_IN;
      CALL  #Timer1 (
           IN                       := #Timer1_IN,
           PT                       := #IN_Alarms_TimeOut,
           Q                        := #Timer1_OUT);
      A     #Timer1_OUT;
      S     #OUT_Alarm_ES_Forward;
NETWORK
TITLE = Allarme Cilindro indietro non segnalato
// Cilindro non tornato in posizione "riposo" in tempo utile
      A     #OUT_EV_Back;
      AN    #OUT_State_CylBack;
      AN    #IN_Hold_Condition;
      A     #IN_Enable;
      =     #Timer2_IN;
      CALL  #Timer2 (
           IN                       := #Timer2_IN,
           PT                       := #IN_Alarms_TimeOut,
           Q                        := #Timer2_OUT);
      A     #Timer2_OUT;
      S     #OUT_Alarm_ES_Back;
NETWORK
TITLE = Allarme Cilindro avanti e indietro entrambi attivi
// Micro contemporanei
      A     #IN_EndStroke_Forward;
      A     #IN_EndStroke_Back;
      A     #IN_Enable;
      S     #OUT_Alarm_ForwBack;
NETWORK
TITLE = Fine
      NOP   0;
NETWORK
TITLE = ALARMS RESET
// Reset allarmi
      A     #IN_Alarms_Reset;
      FP    #FP_ResetAllarmi;
      R     #OUT_Alarm_ES_Forward;
      R     #OUT_Alarm_ES_Back;
      R     #OUT_Alarm_ForwBack;
END_FUNCTION_BLOCK

FUNCTION_BLOCK "Op10.Cycle.General"	// FB 120
VERSION : 0.1
VAR_INPUT
  IN_Cm_ON : BOOL ;	//1: Attiva il ciclo; 0: Reset del ciclo
  IN_HOLD : BOOL ;	//Blocca il ciclo nel passo successivo
  IN_STEP : BOOL ;
END_VAR
VAR_OUTPUT
  OUT_St_CicloInCorso : BOOL ;
  OUT_St_CicloTerminatoOK : BOOL ;
  OUT_St_CicloTerminatoKO : BOOL ;
  OUT_CicloStato : INT ;
  OUT_Page : INT ;
  OUT_Message : INT ;
END_VAR
VAR
  Stato : INT ;
  StatoSeguente : INT ;
  FrontePassoSingolo : BOOL ;
  Stat_CicloTermOk : BOOL ;
  Stat_CicloTermKO : BOOL ;
  Stat_CicloInCorso : BOOL ;
  Timer_Pennarello : SFB 4;
END_VAR
VAR_TEMP
  Pag_Active : ARRAY  [0 .. 100 ] OF BOOL ;
END_VAR
BEGIN
NETWORK
TITLE = FLOW CHART
NETWORK
TITLE = Update state
      A     #IN_Cm_ON;
      JC    M002;
      L     0;
      T     #Stato;
      T     #StatoSeguente;
M002: NOP   0;
//->Update State
      A     #IN_STEP;
      FP    #FrontePassoSingolo;
      ON    #IN_HOLD;	//se usassi UN l'Hold agirebbe anche su avanzamento a passo singolo 
      JCN   N100;
      L     #StatoSeguente;
      T     #Stato;
N100: NOP   0;
// determinazione bit di stato
      CALL  "Conv_INT->BIT" (
           Valore                   := #Stato,
           States                   := "Op10.Cycles".General.State.State_Bit);
NETWORK
TITLE = Detect page active from OP
// serve??????
//      CALL  "Conv_INT->BIT"
//       Valore:=DB325.DBW2
//       States:=#Pag_Active
NETWORK
TITLE = States particular
      L     #Stato;
      L     0;
      <>I;
//->Evita ritardi
      A     #IN_Cm_ON;
      =     #Stat_CicloInCorso;
      A     "Op10.Cycles".General.State.State_Bit[60];
      =     #Stat_CicloTermOk;
      A     "Op10.Cycles".Restore.State.State_Bit[63];
      =     #Stat_CicloTermKO;
NETWORK
TITLE = Diagnostic default
//    L     0
//    T     #Page
//    L     0
//    T     #Message 
//      L     6
//      T     #StatoSeguente
NETWORK
TITLE = State <0>: Ciclo off
      A     "Op10.Cycles".General.State.State_Bit[0];
      A     #IN_Cm_ON;
      JC    A000;
      L     "Op10.Cycles".General.State.Page;
      T     #OUT_Page;
      L     1;	// Ciclo off
      T     #OUT_Message;
      JU    Z000;
A000: L     10;
      T     #StatoSeguente;
Z000: NOP   0;
NETWORK
TITLE = State <10>: Inserimento pezzi su attrezzo e start ciclo
      A     "Op10.Cycles".General.State.State_Bit[10];
      JCN   Z010;
      A     "Op10.Bench.MapE".Sblocco_pezzo_Su;
      A     "Op10.Bench.MapE".Index_cassetto_Su;
      A     "Op10.Tools.MapE".Presenza_nozzle_ring;
      O     "Op10.Bench.Recipe".Disable.CkPresenzaNozzleRing;
      A(;
      A     "Op10.Tools.MapE".Spacer_1_presente;
      AN    "Op10.Tools.MapE".Spacer_1_invertito;
      O     "Op10.Bench.Recipe".Disable.CkPresenzaSpacer1;
      );
      A(;
      A     "Op10.Tools.MapE".Spacer_2_presente;
      AN    "Op10.Tools.MapE".Spacer_2_invertito;
      O     "Op10.Bench.Recipe".Disable.CkPresenzaSpacer2;
      );
      A(;
      A     "Op10.Tools.MapE".Spacer_3_presente;
      AN    "Op10.Tools.MapE".Spacer_3_invertito;
      O     "Op10.Bench.Recipe".Disable.CkPresenzaSpacer3;
      );
      A     "Op10.Bench.Systems".Command.FP_Consenso_operatore;
      JC    Y010;
// Messaggi
// Inserisci spacer correttamente          
      A(;
      AN    "Op10.Tools.MapE".Spacer_1_presente;
      AN    "Op10.Bench.Recipe".Disable.CkPresenzaSpacer1;
      );
      O(;
      AN    "Op10.Tools.MapE".Spacer_2_presente;
      AN    "Op10.Bench.Recipe".Disable.CkPresenzaSpacer2;
      );
      O(;
      AN    "Op10.Tools.MapE".Spacer_3_presente;
      AN    "Op10.Bench.Recipe".Disable.CkPresenzaSpacer3;
      );
      JC    A010;
// almeno uno Spacer inserito male
      A(;
      A     "Op10.Tools.MapE".Spacer_1_invertito;
      AN    "Op10.Bench.Recipe".Disable.CkPresenzaSpacer1;
      );
      O(;
      A     "Op10.Tools.MapE".Spacer_2_invertito;
      AN    "Op10.Bench.Recipe".Disable.CkPresenzaSpacer2;
      );
      O(;
      A     "Op10.Tools.MapE".Spacer_2_invertito;
      AN    "Op10.Bench.Recipe".Disable.CkPresenzaSpacer3;
      );
      JC    B010;
// Inserisci nozzle ring
      AN    "Op10.Tools.MapE".Presenza_nozzle_ring;
      AN    "Op10.Bench.Recipe".Disable.CkPresenzaNozzleRing;
      JC    C010;
// Start ciclo per Bloccare il pezzo
      JU    D010;
A010: L     "Op10.Cycles".General.State.Page;
      T     #OUT_Page;
      L     2;	// Inserisci spacer correttamente
      T     #OUT_Message;
      JU    Z010;
B010: L     "Op10.Cycles".General.State.Page;
      T     #OUT_Page;
      L     3;	// almeno uno Spacer inserito male
      T     #OUT_Message;
      JU    Z010;
C010: L     "Op10.Cycles".General.State.Page;
      T     #OUT_Page;
      L     4;	// Inserisci nozzle ring
      T     #OUT_Message;
      JU    Z010;
D010: L     "Op10.Cycles".General.State.Page;
      T     #OUT_Page;
      L     5;	// Start ciclo per Bloccare il pezzo
      T     #OUT_Message;
      JU    Z010;
// Stati di destinazione
Y010: L     13;
      T     #StatoSeguente;
Z010: NOP   0;
NETWORK
TITLE = State <13>: Blocca Pezzo e sblocca index
      A     "Op10.Cycles".General.State.State_Bit[13];
      A     "Op10.Bench.Systems".State.Cassetto_dentro;
      L     S5T#500MS;
      SD    "OP10St13_Cassetto_dentro";
      A     "Op10.Cycles".General.State.State_Bit[13];
      JCN   Z013;
      A     "Op10.Bench.MapE".Sblocco_pezzo_Giu;
      A     "Op10.Bench.MapE".Index_cassetto_Giu;
      A(;
      A     "Op10.Bench.Systems".State.Ribaditrice_alta;
      O     "Op10.Bench.Systems".State._Ribad_in_fuori_ingombro;
      );
      A     "OP10St13_Cassetto_dentro";
      JC    Y013;
// Messaggi
// Blocco pezzo e sblocco cassetto in corso
      AN    "Op10.Bench.MapE".Sblocco_pezzo_Giu;
      ON    "Op10.Bench.MapE".Index_cassetto_Giu;
      JC    A013;
// Porta cassetto in zona di lavorazione
      AN    "Op10.Bench.Systems".State.Cassetto_dentro;
      JC    B013;
      JU    B013;
A013: L     "Op10.Cycles".General.State.Page;
      T     #OUT_Page;
      L     6;	// Blocco pezzo e sblocco cassetto in corso
      T     #OUT_Message;
      JU    Z013;
B013: L     "Op10.Cycles".General.State.Page;
      T     #OUT_Page;
      L     7;	// Porta cassetto in zona di lavorazione
      T     #OUT_Message;
      JU    Z013;
// Stati di destinazione
Y013: L     16;
      T     #StatoSeguente;
Z013: NOP   0;
NETWORK
TITLE = State <16>: Blocca cassetto e prenota ribaditrice
      A     "Op10.Cycles".General.State.State_Bit[16];
      JCN   Z016;
      A     "Op10.Bench.MapE".Sblocco_pezzo_Giu;
      A     "Op10.Bench.MapE".Index_cassetto_Su;
      A     "Op10.Bench.Systems".State.Cassetto_dentro;
      A     "Op10.Bench.Systems".State._Ribaditrice_a_disposiz;
      JC    Y016;
// Messaggi
// Blocco cassetto in corso
      AN    "Op10.Bench.MapE".Sblocco_pezzo_Giu;
      ON    "Op10.Bench.MapE".Index_cassetto_Su;
      ON    "Op10.Bench.Systems".State.Cassetto_dentro;
      JC    A016;
// Attesa prenotazione ribaditrice
      AN    "Op10.Bench.Systems".State._Ribaditrice_a_disposiz;
      JC    B016;
      JU    B016;
A016: L     "Op10.Cycles".General.State.Page;
      T     #OUT_Page;
      L     8;	// Blocco cassetto in corso
      T     #OUT_Message;
      JU    Z016;
B016: L     "Op10.Cycles".General.State.Page;
      T     #OUT_Page;
      L     9;	//  Attesa prenotazione ribaditrice
      T     #OUT_Message;
      JU    Z016;
// Stati di destinazione
Y016: L     20;
      T     #StatoSeguente;
Z016: NOP   0;
NETWORK
TITLE = State <20>: Vai a quota di ribaditura punto corrente
      A     "Op10.Cycles".General.State.State_Bit[20];
      JCN   Z020;
      A     "Op10.Bench.Systems".State._Assi_posiz_raggiunta;
      A     "Op10.Bench.Systems".State.Ribaditrice_in_marcia;
      JC    Y020;
// Messaggi
// Posizionamento assi
      L     "Op10.Cycles".General.State.Page;
      T     #OUT_Page;
      L     14;	// Posizionamento assi
      T     #OUT_Message;
      JU    Z020;
// Stati di destinazione
Y020: L     25;
      T     #StatoSeguente;
Z020: NOP   0;
NETWORK
TITLE = State <25>: Esegui ribaditura punto corrente
      A     "Op10.Cycles".General.State.State_Bit[25];
      JCN   Z025;
      A     "Op10.Bench.Systems".State.Ribaditura_effettuata;
      JC    Y025;
// Messaggi
// Ribaditura spacer in corso
      L     "Op10.Cycles".General.State.Page;
      T     #OUT_Page;
      L     9;	// Ribaditura spacer in corso
      T     #OUT_Message;
      JU    Z025;
// Stati di destinazione
Y025: L     30;
      T     #StatoSeguente;
Z025: NOP   0;
NETWORK
TITLE = State <30>: Risali ribaditrice
      A     "Op10.Cycles".General.State.State_Bit[30];
      JCN   Z030;
      A     "Op10.Bench.Systems".State.Ribaditrice_alta;
      A(;
      L     "Op10.Bench.Systems".Data.Num_punto_in_lavorazione;
      L     "Op10.Bench.Recipe".NumeroPosizioni;
      <I;
      );
      JC    Y030;
      A     "Op10.Bench.Systems".State.Ribaditrice_alta;
      A(;
      L     "Op10.Bench.Systems".Data.Num_punto_in_lavorazione;
      L     "Op10.Bench.Recipe".NumeroPosizioni;
      >=I;
      );
      JC    X030;
// Messaggi
// Ribaditura spacer in corso
      L     "Op10.Cycles".General.State.Page;
      T     #OUT_Page;
      L     9;	// Ribaditura spacer in corso
      T     #OUT_Message;
      JU    Z030;
// Stati di destinazione
Y030: L     20;
      T     #StatoSeguente;
      JU    Z030;
X030: L     35;
      T     #StatoSeguente;
Z030: NOP   0;
NETWORK
TITLE = State <35>: Sblocco index e cassetto fuori
      A     "Op10.Cycles".General.State.State_Bit[35];
      A     "Op10.Bench.Systems".State.Cassetto_fuori;
      L     S5T#500MS;
      SD    "OP10St35_Cassetto_fuori";
      A     "Op10.Cycles".General.State.State_Bit[35];
      JCN   Z035;
      A     "Op10.Bench.MapE".Index_cassetto_Giu;
      A     "OP10St35_Cassetto_fuori";
      JC    Y035;
// Messaggi
// Sblocco index in corso
      AN    "Op10.Bench.MapE".Index_cassetto_Giu;
      JC    A035;
// Porta cassetto in zona di carico
      JU    B035;
A035: L     "Op10.Cycles".General.State.Page;
      T     #OUT_Page;
      L     10;	// Sblocco index in corso
      T     #OUT_Message;
      JU    Z035;
B035: L     "Op10.Cycles".General.State.Page;
      T     #OUT_Page;
      L     11;	// Porta cassetto in zona di carico
      T     #OUT_Message;
      JU    Z035;
// Stati di destinazione
Y035: L     40;
      T     #StatoSeguente;
Z035: NOP   0;
NETWORK
TITLE = State <40>: Sblocco pezzo e fine lavorazione
      A     "Op10.Cycles".General.State.State_Bit[40];
      JCN   Z040;
      A     "Op10.Bench.MapE".Index_cassetto_Su;
      A     "Op10.Bench.MapE".Sblocco_pezzo_Su;
      A     "Op10.Bench.Systems".State.Cassetto_fuori;
      A(;
      AN    "Op10.Tools.MapE".Presenza_nozzle_ring;
      O     "Op10.Bench.Recipe".Disable.CkPresenzaNozzleRing;
      );
      A(;
      AN    "Op10.Tools.MapE".Spacer_1_presente;
      O     "Op10.Bench.Recipe".Disable.CkPresenzaSpacer1;
      );
      A(;
      AN    "Op10.Tools.MapE".Spacer_2_presente;
      O     "Op10.Bench.Recipe".Disable.CkPresenzaSpacer2;
      );
      A(;
      AN    "Op10.Tools.MapE".Spacer_3_presente;
      O     "Op10.Bench.Recipe".Disable.CkPresenzaSpacer3;
      );
      JC    Y040;
// Messaggi
// Blocco index e sblocco pezzo in corso
      AN    "Op10.Bench.MapE".Index_cassetto_Su;
      ON    "Op10.Bench.MapE".Sblocco_pezzo_Su;
      JC    A040;
// Rimuovi pezzo buono dalla stazione
      JU    B040;
A040: L     "Op10.Cycles".General.State.Page;
      T     #OUT_Page;
      L     12;	// Blocco index e sblocco pezzo in corso
      T     #OUT_Message;
      JU    Z040;
B040: L     "Op10.Cycles".General.State.Page;
      T     #OUT_Page;
      L     13;	// Rimuovi pezzo buono dalla stazione
      T     #OUT_Message;
      JU    Z040;
// Stati di destinazione
Y040: L     60;
      T     #StatoSeguente;
Z040: NOP   0;
NETWORK
TITLE =
      A     "Op10.Cycles".General.State.State_Bit[60];
      JCN   Z060;
// Stati di destinazione
      L     10;
      T     #StatoSeguente;
Z060: NOP   0;
NETWORK
TITLE = Output
      L     #Stato;
      T     #OUT_CicloStato;
      A     #Stat_CicloInCorso;
      =     #OUT_St_CicloInCorso;
      A     #Stat_CicloTermOk;
      =     #OUT_St_CicloTerminatoOK;
      A     #Stat_CicloTermKO;
      =     #OUT_St_CicloTerminatoKO;
END_FUNCTION_BLOCK

FUNCTION_BLOCK "Op10.Cycle.Restore"	// FB 121
VERSION : 0.1
VAR_INPUT
  IN_Cm_ON : BOOL ;	//1: Attiva il ciclo; 0: Reset del ciclo
  IN_HOLD : BOOL ;	//Blocca il ciclo nel passo successivo
  IN_STEP : BOOL ;
END_VAR
VAR_OUTPUT
  OUT_St_CicloInCorso : BOOL ;
  OUT_St_CicloTerminatoOK : BOOL ;
  OUT_St_CicloTerminatoKO : BOOL ;
  OUT_CicloStato : INT ;
  OUT_Page : INT ;
  OUT_Message : INT ;
END_VAR
VAR
  Stato : INT ;
  StatoSeguente : INT ;
  FrontePassoSingolo : BOOL ;
  Stat_CicloTermOk : BOOL ;
  Stat_CicloTermKO : BOOL ;
  Stat_CicloInCorso : BOOL ;
  Timer_Pennarello : SFB 4;
END_VAR
VAR_TEMP
  Pag_Active : ARRAY  [0 .. 100 ] OF BOOL ;
END_VAR
BEGIN
NETWORK
TITLE = FLOW CHART
NETWORK
TITLE = Update state
      A     #IN_Cm_ON;
      JC    M002;
      L     0;
      T     #Stato;
      T     #StatoSeguente;
M002: NOP   0;
//->Update State
      A     #IN_STEP;
      FP    #FrontePassoSingolo;
      ON    #IN_HOLD;	//se usassi UN l'Hold agirebbe anche su avanzamento a passo singolo 
      JCN   N100;
      L     #StatoSeguente;
      T     #Stato;
N100: NOP   0;
// determinazione bit di stato
      CALL  "Conv_INT->BIT" (
           Valore                   := #Stato,
           States                   := "Op10.Cycles".Restore.State.State_Bit);
NETWORK
TITLE = States particular
      L     #Stato;
      L     0;
      <>I;
//->Evita ritardi
      A     #IN_Cm_ON;
      =     #Stat_CicloInCorso;
      A     "Op10.Cycles".Restore.State.State_Bit[60];
      =     #Stat_CicloTermOk;
      A     "Op10.Cycles".Restore.State.State_Bit[63];
      =     #Stat_CicloTermKO;
NETWORK
TITLE = State <0>: Ciclo off
      A     "Op10.Cycles".Restore.State.State_Bit[0];
      A     #IN_Cm_ON;
      JC    A000;
      L     "Op10.Cycles".Restore.State.Page;
      T     #OUT_Page;
      L     20;	// ciclo off
      T     #OUT_Message;
      JU    Z000;
A000: L     10;
      T     #StatoSeguente;
Z000: NOP   0;
NETWORK
TITLE = State <10>: Sali ribaditrice
      A     "Op10.Cycles".Restore.State.State_Bit[10];
      JCN   Z010;
      A     "Op10.Bench.Systems".State.Ribaditrice_alta;
      O     "Op10.Bench.Systems".State._Ribad_in_fuori_ingombro;
      AN    "Op10.Bench.MapE".Cassetto_fuori;
      JC    Y010;
      A     "Op10.Bench.Systems".State.Ribaditrice_alta;
      O     "Op10.Bench.Systems".State._Ribad_in_fuori_ingombro;
      A     "Op10.Bench.MapE".Cassetto_fuori;
      JC    X010;
// Messaggi
// Salita ribaditrice in corso
      L     "Op10.Cycles".Restore.State.Page;
      T     #OUT_Page;
      L     21;	// Salita ribaditrice in corso
      T     #OUT_Message;
      JU    Z010;
// Stati di destinazione
Y010: L     15;
      T     #StatoSeguente;
      JU    Z010;
X010: L     20;
      T     #StatoSeguente;
Z010: NOP   0;
NETWORK
TITLE = State <15>: Sblocca index e cassetto fuori
      A     "Op10.Cycles".Restore.State.State_Bit[15];
      A     "Op10.Bench.Systems".State.Cassetto_fuori;
      L     S5T#500MS;
      SD    "RP10St15_Cassetto_fuori";
      A     "Op10.Cycles".Restore.State.State_Bit[15];
      JCN   Z015;
      A     "Op10.Bench.MapE".Index_cassetto_Giu;
      A     "RP10St15_Cassetto_fuori";
      JC    Y015;
// Messaggi
//   Sblocco index in corso
      AN    "Op10.Bench.MapE".Index_cassetto_Giu;
      JC    A015;
// Porta cassetto in zona di scarico
      JU    B015;
A015: L     "Op10.Cycles".Restore.State.Page;
      T     #OUT_Page;
      L     22;	//  Sblocco index in corso
      T     #OUT_Message;
      JU    Z015;
B015: L     "Op10.Cycles".Restore.State.Page;
      T     #OUT_Page;
      L     23;	// Porta cassetto in zona di scarico
      T     #OUT_Message;
      JU    Z015;
// Stati di destinazione
Y015: L     20;
      T     #StatoSeguente;
Z015: NOP   0;
NETWORK
TITLE = State <20>: Blocca index e sblocca pezzo - rimuovi scarto
      A     "Op10.Cycles".Restore.State.State_Bit[20];
      JCN   Z020;
      A     "Op10.Bench.MapE".Sblocco_pezzo_Su;
      A     "Op10.Bench.MapE".Index_cassetto_Su;
      A     "Op10.Bench.Systems".State.Cassetto_fuori;
      A(;
      AN    "Op10.Tools.MapE".Presenza_nozzle_ring;
      O     "Op10.Bench.Recipe".Disable.CkPresenzaNozzleRing;
      );
      JC    Y020;
// Messaggi
// Blocco index e sblocco pezzo in corso
      AN    "Op10.Bench.MapE".Sblocco_pezzo_Su;
      ON    "Op10.Bench.MapE".Index_cassetto_Su;
      ON    "Op10.Bench.Systems".State.Cassetto_fuori;
      JC    A020;
// Rimuovi pezzo scarto dalla stazione
      JU    B020;
A020: L     "Op10.Cycles".Restore.State.Page;
      T     #OUT_Page;
      L     24;	// Blocco index e sblocco pezzo in corso
      T     #OUT_Message;
      JU    Z020;
B020: L     "Op10.Cycles".Restore.State.Page;
      T     #OUT_Page;
      L     25;	// Rimuovi pezzo scarto dalla stazione
      T     #OUT_Message;
      JU    Z020;
// Stati di destinazione
Y020: L     60;
      T     #StatoSeguente;
Z020: NOP   0;
NETWORK
TITLE = Output
      L     #Stato;
      T     #OUT_CicloStato;
      A     #Stat_CicloInCorso;
      =     #OUT_St_CicloInCorso;
      A     #Stat_CicloTermOk;
      =     #OUT_St_CicloTerminatoOK;
      A     #Stat_CicloTermKO;
      =     #OUT_St_CicloTerminatoKO;
END_FUNCTION_BLOCK

FUNCTION_BLOCK "Op20.Cycle.General"	// FB 170
VERSION : 0.1
VAR_INPUT
  IN_Cm_ON : BOOL ;	//1: Attiva il ciclo; 0: Reset del ciclo
  IN_HOLD : BOOL ;	//Blocca il ciclo nel passo successivo
  IN_STEP : BOOL ;
END_VAR
VAR_OUTPUT
  OUT_St_CicloInCorso : BOOL ;
  OUT_St_CicloTerminatoOK : BOOL ;
  OUT_St_CicloTerminatoKO : BOOL ;
  OUT_CicloStato : INT ;
  OUT_Page : INT ;
  OUT_Message : INT ;
END_VAR
VAR
  Stato : INT ;
  StatoSeguente : INT ;
  FrontePassoSingolo : BOOL ;
  Stat_CicloTermOk : BOOL ;
  Stat_CicloTermKO : BOOL ;
  Stat_CicloInCorso : BOOL ;
END_VAR
VAR_TEMP
  Pag_Active : ARRAY  [0 .. 100 ] OF BOOL ;
END_VAR
BEGIN
NETWORK
TITLE = FLOW CHART
NETWORK
TITLE = Update state
      A     #IN_Cm_ON;
      JC    M002;
      L     0;
      T     #Stato;
      T     #StatoSeguente;
M002: NOP   0;
//->Update State
      A     #IN_STEP;
      FP    #FrontePassoSingolo;
      ON    #IN_HOLD;	//se usassi UN l'Hold agirebbe anche su avanzamento a passo singolo 
      JCN   N100;
      L     #StatoSeguente;
      T     #Stato;
N100: NOP   0;
// determinazione bit di stato
      CALL  "Conv_INT->BIT" (
           Valore                   := #Stato,
           States                   := "Op20.Cycles".General.State.State_Bit);
NETWORK
TITLE = States particular
      L     #Stato;
      L     0;
      <>I;
//->Evita ritardi
      A     #IN_Cm_ON;
      =     #Stat_CicloInCorso;
      A     "Op20.Cycles".General.State.State_Bit[60];
      =     #Stat_CicloTermOk;
      A     "Op20.Cycles".Restore.State.State_Bit[63];
      =     #Stat_CicloTermKO;
NETWORK
TITLE = Diagnostic default
NETWORK
TITLE = State <0>: Ciclo off
      A     "Op20.Cycles".General.State.State_Bit[0];
      A     #IN_Cm_ON;
      JC    A000;
      L     "Op20.Cycles".General.State.Page;
      T     #OUT_Page;
      L     1;	// Ciclo off
      T     #OUT_Message;
      JU    Z000;
A000: L     10;
      T     #StatoSeguente;
Z000: NOP   0;
NETWORK
TITLE = State <10>: Inserimento pezzi su attrezzo e cassetto dentrro
      A     "Op20.Bench.MapE".Cassetto_dentro;
      L     S5T#500MS;
      SD    "OP20ST10_Cassetto_dentro";
      A     "OP20ST10_Cassetto_dentro";
      FP    "AppoFP_M52.0";
      =     "Op20.Bench.Systems".State.FP_Cassettodentro;
      A     "Op20.Bench.Systems".State.FP_Cassettodentro;
      A     "Op20.Cycles".General.State.State_Bit[10];
      S     "Op20.Bench.Systems".State.CassetDentroInizioCiclo;
      A     "Op20.Bench.Systems".State.CassetDentroInizioCiclo;
      AN    "Op20.Bench.MapE".Cassetto_dentro;
      ON    "Op20.Cycles".General.State.State_Bit[10];
      R     "Op20.Bench.Systems".State.CassetDentroInizioCiclo;
      A     "Op20.Bench.Systems".State.CassetDentroInizioCiclo;
      L     S5T#500MS;
      SD    "TOP20_Cassetto dentro";
      A     "Op20.Cycles".General.State.State_Bit[10];
      JCN   Z010;
      A     "TOP20_Cassetto dentro";
      JC    Y010;
// Messaggi
// Inserisci pezzi e porta cassetto dentro
      L     "Op20.Cycles".General.State.Page;
      T     #OUT_Page;
      L     2;	//  Inserisci pezzi e porta cassetto dentro
      T     #OUT_Message;
      JU    Z010;
// Stati di destinazione
Y010: L     15;
      T     #StatoSeguente;
Z010: NOP   0;
NETWORK
TITLE = State <15>: Blocca cassetto dentrro
      A     "Op20.Cycles".General.State.State_Bit[15];
      JCN   Z015;
      A     "Op20.Bench.MapE".Cassetto_dentro;
      A     "Op20.Bench.MapE".Index_cassetto_Su;
      JC    Y015;
// Messaggi
// Blocco cassetto in corso
      L     "Op20.Cycles".General.State.Page;
      T     #OUT_Page;
      L     3;	// Blocco cassetto in corso
      T     #OUT_Message;
      JU    Z015;
// Stati di destinazione
Y015: L     20;
      T     #StatoSeguente;
Z015: NOP   0;
NETWORK
TITLE = State <20>: Discesa gruppo di piantaggio
      A     "Op20.Cycles".General.State.State_Bit[20];
      JCN   Z020;
      A     "Op20.Bench.MapE".Gruppo_piantaggio_Giu;
      JC    Y020;
// Messaggi
// Discesa gruppo di piantaggio
      L     "Op20.Cycles".General.State.Page;
      T     #OUT_Page;
      L     4;	// Discesa gruppo di piantaggio
      T     #OUT_Message;
      JU    Z020;
// Stati di destinazione
Y020: L     25;
      T     #StatoSeguente;
Z020: NOP   0;
NETWORK
TITLE = State <25>: Discesa piantaggio
      A     "Op20.Cycles".General.State.State_Bit[25];
      JCN   Z025;
      A     "Op20.Bench.Systems".State.Piantaggiofinito;
      JC    Y025;
// Messaggi
// Piantaggio in corso
      L     "Op20.Cycles".General.State.Page;
      T     #OUT_Page;
      L     5;	// Piantaggio in corso
      T     #OUT_Message;
      JU    Z025;
// Stati di destinazione
Y025: L     30;
      T     #StatoSeguente;
Z025: NOP   0;
NETWORK
TITLE = State <30>: Risalita piantaggio
      A     "Op20.Cycles".General.State.State_Bit[30];
      JCN   Z030;
      A     "Op20.Bench.MapE".Gruppo_piantaggio_Su;
      A     "Op20.Bench.MapE".Piantaggio_Su;
      JC    Y030;
// Messaggi
// Risalita pressa in corso
      L     "Op20.Cycles".General.State.Page;
      T     #OUT_Page;
      L     6;	// Risalita pressa in corso
      T     #OUT_Message;
      JU    Z030;
// Stati di destinazione
Y030: L     35;
      T     #StatoSeguente;
Z030: NOP   0;
NETWORK
TITLE = State <35>: Sblocco cassetto
      A     "Op20.Cycles".General.State.State_Bit[35];
      JCN   Z035;
      A     "Op20.Bench.MapE".Index_cassetto_Giu;
      JC    Y035;
// Messaggi
// Sblocco cassetto in corso
      L     "Op20.Cycles".General.State.Page;
      T     #OUT_Page;
      L     7;	// Sblocco cassetto in corso
      T     #OUT_Message;
      JU    Z035;
// Stati di destinazione
Y035: L     60;
      T     #StatoSeguente;
Z035: NOP   0;
NETWORK
TITLE =
      A     "Op20.Cycles".General.State.State_Bit[60];
      JCN   Z060;
      L     10;
      T     #StatoSeguente;
Z060: NOP   0;
NETWORK
TITLE = Output
      L     #Stato;
      T     #OUT_CicloStato;
      A     #Stat_CicloInCorso;
      =     #OUT_St_CicloInCorso;
      A     #Stat_CicloTermOk;
      =     #OUT_St_CicloTerminatoOK;
      A     #Stat_CicloTermKO;
      =     #OUT_St_CicloTerminatoKO;
END_FUNCTION_BLOCK

FUNCTION_BLOCK "Op20.Cycle.Restore"	// FB 171
VERSION : 0.1
VAR_INPUT
  IN_Cm_ON : BOOL ;	//1: Attiva il ciclo; 0: Reset del ciclo
  IN_HOLD : BOOL ;	//Blocca il ciclo nel passo successivo
  IN_STEP : BOOL ;
END_VAR
VAR_OUTPUT
  OUT_St_CicloInCorso : BOOL ;
  OUT_St_CicloTerminatoOK : BOOL ;
  OUT_St_CicloTerminatoKO : BOOL ;
  OUT_CicloStato : INT ;
  OUT_Page : INT ;
  OUT_Message : INT ;
END_VAR
VAR
  Stato : INT ;
  StatoSeguente : INT ;
  FrontePassoSingolo : BOOL ;
  Stat_CicloTermOk : BOOL ;
  Stat_CicloTermKO : BOOL ;
  Stat_CicloInCorso : BOOL ;
END_VAR
VAR_TEMP
  Pag_Active : ARRAY  [0 .. 100 ] OF BOOL ;
END_VAR
BEGIN
NETWORK
TITLE = FLOW CHART
NETWORK
TITLE = Update state
      A     #IN_Cm_ON;
      JC    M002;
      L     0;
      T     #Stato;
      T     #StatoSeguente;
M002: NOP   0;
//->Update State
      A     #IN_STEP;
      FP    #FrontePassoSingolo;
      ON    #IN_HOLD;	//se usassi UN l'Hold agirebbe anche su avanzamento a passo singolo 
      JCN   N100;
      L     #StatoSeguente;
      T     #Stato;
N100: NOP   0;
// determinazione bit di stato
      CALL  "Conv_INT->BIT" (
           Valore                   := #Stato,
           States                   := "Op20.Cycles".Restore.State.State_Bit);
NETWORK
TITLE = States particular
      L     #Stato;
      L     0;
      <>I;
//->Evita ritardi
      A     #IN_Cm_ON;
      =     #Stat_CicloInCorso;
      A     "Op20.Cycles".Restore.State.State_Bit[60];
      =     #Stat_CicloTermOk;
      A     "Op20.Cycles".Restore.State.State_Bit[63];
      =     #Stat_CicloTermKO;
NETWORK
TITLE = Diagnostic default
NETWORK
TITLE = State <0>: Ciclo off
      A     "Op20.Cycles".Restore.State.State_Bit[0];
      A     #IN_Cm_ON;
      JC    A000;
      L     "Op20.Cycles".Restore.State.Page;
      T     #OUT_Page;
      L     1;	// Ciclo off
      T     #OUT_Message;
      JU    Z000;
A000: L     10;
      T     #StatoSeguente;
Z000: NOP   0;
NETWORK
TITLE = State <10>: Risalita piantaggio
      A     "Op20.Cycles".Restore.State.State_Bit[10];
      JCN   Z010;
      A     "Op20.Bench.MapE".Gruppo_piantaggio_Su;
      A     "Op20.Bench.MapE".Piantaggio_Su;
      JC    Y010;
// Messaggi
// Risalita pressa in corso
      L     "Op20.Cycles".Restore.State.Page;
      T     #OUT_Page;
      L     6;	// Risalita pressa in corso
      T     #OUT_Message;
      JU    Z010;
// Stati di destinazione
Y010: L     15;
      T     #StatoSeguente;
Z010: NOP   0;
NETWORK
TITLE = State <15>: Sblocco cassetto
      A     "Op20.Cycles".Restore.State.State_Bit[15];
      JCN   Z015;
      A     "Op20.Bench.MapE".Index_cassetto_Giu;
      JC    Y015;
// Messaggi
// Sblocco cassetto in corso
      L     "Op20.Cycles".Restore.State.Page;
      T     #OUT_Page;
      L     7;	// Sblocco cassetto in corso
      T     #OUT_Message;
      JU    Z015;
// Stati di destinazione
Y015: L     60;
      T     #StatoSeguente;
Z015: NOP   0;
NETWORK
TITLE = Output
      L     #Stato;
      T     #OUT_CicloStato;
      A     #Stat_CicloInCorso;
      =     #OUT_St_CicloInCorso;
      A     #Stat_CicloTermOk;
      =     #OUT_St_CicloTerminatoOK;
      A     #Stat_CicloTermKO;
      =     #OUT_St_CicloTerminatoKO;
END_FUNCTION_BLOCK

FUNCTION_BLOCK "Op40.Cycle.General"	// FB 220
VERSION : 0.1
VAR_INPUT
  IN_Cm_ON : BOOL ;	//1: Attiva il ciclo; 0: Reset del ciclo
  IN_HOLD : BOOL ;	//Blocca il ciclo nel passo successivo
  IN_STEP : BOOL ;
END_VAR
VAR_OUTPUT
  OUT_St_CicloInCorso : BOOL ;
  OUT_St_CicloTerminatoOK : BOOL ;
  OUT_St_CicloTerminatoKO : BOOL ;
  OUT_CicloStato : INT ;
  OUT_Page : INT ;
  OUT_Message : INT ;
END_VAR
VAR
  Stato : INT ;
  StatoSeguente : INT ;
  FrontePassoSingolo : BOOL ;
  Stat_CicloTermOk : BOOL ;
  Stat_CicloTermKO : BOOL ;
  Stat_CicloInCorso : BOOL ;
  Timer_Pennarello : SFB 4;
END_VAR
VAR_TEMP
  Pag_Active : ARRAY  [0 .. 100 ] OF BOOL ;
END_VAR
BEGIN
NETWORK
TITLE = FLOW CHART
NETWORK
TITLE = Update state
      A     #IN_Cm_ON;
      JC    M002;
      L     0;
      T     #Stato;
      T     #StatoSeguente;
M002: NOP   0;
//->Update State
      A     #IN_STEP;
      FP    #FrontePassoSingolo;
      ON    #IN_HOLD;	//se usassi UN l'Hold agirebbe anche su avanzamento a passo singolo 
      JCN   N100;
      L     #StatoSeguente;
      T     #Stato;
N100: NOP   0;
// determinazione bit di stato
      CALL  "Conv_INT->BIT" (
           Valore                   := #Stato,
           States                   := "Op40.Cycles".General.State.State_Bit);
NETWORK
TITLE = States particular
      L     #Stato;
      L     0;
      <>I;
//->Evita ritardi
      A     #IN_Cm_ON;
      =     #Stat_CicloInCorso;
      A     "Op40.Cycles".General.State.State_Bit[60];
      =     #Stat_CicloTermOk;
      A     "Op40.Cycles".General.State.State_Bit[63];
      =     #Stat_CicloTermKO;
NETWORK
TITLE = Diagnostic default
//    L     0
//    T     #Page
//    L     0
//    T     #Message 
//      L     6
//      T     #StatoSeguente
NETWORK
TITLE = State <0>: Ciclo off
      A     "Op40.Cycles".General.State.State_Bit[0];
      A     #IN_Cm_ON;
      JC    A000;
      L     "Op10.Cycles".Restore.State.Page;
      T     #OUT_Page;
      L     1;	// ciclo off
      T     #OUT_Message;
      JU    Z000;
A000: L     10;
      T     #StatoSeguente;
Z000: NOP   0;
NETWORK
TITLE = State <10>: Inserimento pezzi su attrezzo e start ciclo
      A     "Op40.Cycles".General.State.State_Bit[10];
      JCN   Z010;
      A     "Op40.Bench.MapE".Unlock_parts_up;
      A     "Op40.Bench.MapE".Box_index_down;
      A     "Op40.Bench.Systems".Command.FP_Consenso_operatore;
      JC    Y010;
// Messaggi
// Inserisci nozzle ring e Start ciclo
      L     "Op40.Cycles".General.State.Page;
      T     #OUT_Page;
      L     4;	// Inserisci nozzle ring e start ciclo
      T     #OUT_Message;
      JU    Z010;
// Stati di destinazione
Y010: L     11;
      T     #StatoSeguente;
Z010: NOP   0;
NETWORK
TITLE = State <11>: Blocca index e controlla presenza pezzo
      A     "Op40.Cycles".General.State.State_Bit[11];
      JCN   Z011;
      A     "Op40.Bench.MapE".Unlock_parts_down;
      A(;
      A     "Op40.Tools.MapE".Presenza_pin_roller;
      O     "Op40.Bench.Recipe".Disable.CkPresenzaNozzleRing;
//     O     "Op40.Bench.Recipe".Disable.CkPresenzaPipe
      );
      JC    Y011;
      A     "Op40.Bench.Systems".Command.FP_Consenso_operatore;
      JC    X011;
// Messaggi
// Inserisci nozzle ring
      AN    "Op40.Tools.MapE".Presenza_pin_roller;
      A     "Op40.Bench.Recipe".Disable.CkPresenzaPipe;
      JC    A011;
      JU    Z011;
A011: L     "Op40.Cycles".General.State.Page;
      T     #OUT_Page;
      L     5;	// Inserisci nozzle ring
      T     #OUT_Message;
      JU    Z011;
// Stati di destinazione
X011: L     10;
      T     #StatoSeguente;
      JU    Z011;
Y011: L     13;
      T     #StatoSeguente;
Z011: NOP   0;
NETWORK
TITLE = State <13>: sblocca index
      A     "Op40.Cycles".General.State.State_Bit[13];
      A     "Op40.Bench.Systems".State.Cassetto_dentro;
      L     S5T#500MS;
      SD    "OP40St13_Cassetto_dentro";
      A     "Op40.Cycles".General.State.State_Bit[13];
      JCN   Z013;
      A     "Op40.Bench.MapE".Unlock_parts_down;
      A     "Op40.Bench.MapE".Box_index_up;
      A(;
      A     "Op40.Bench.Systems".State.Ribaditrice_alta;
      O     "Op40.Bench.Systems".State._Ribad_in_fuori_ingombro;
      );
      A     "OP40St13_Cassetto_dentro";
      A     "Op40.Bench.MapE".Pipe_placed;
      A     "Op40.Bench.MapE".Ring_lock_pipe_present;
      JC    Y013;
// Messaggi
// Blocco pezzo e sblocco cassetto in corso
      AN    "Op40.Bench.MapE".Unlock_parts_down;
      ON    "Op40.Bench.MapE".Box_index_up;
      JC    A013;
// Porta cassetto in zona di lavorazione
      AN    "Op40.Bench.Systems".State.Cassetto_dentro;
      JC    B013;
      JU    C013;
A013: L     "Op40.Cycles".General.State.Page;
      T     #OUT_Page;
      L     6;	// Blocco pezzo e sblocco cassetto in corso
      T     #OUT_Message;
      JU    Z013;
B013: L     "Op40.Cycles".General.State.Page;
      T     #OUT_Page;
      L     7;	// Porta cassetto in zona di lavorazione
      T     #OUT_Message;
      JU    Z013;
C013: L     "Op40.Cycles".General.State.Page;
      T     #OUT_Page;
      L     3;	// Controlla presenza Pipe
      T     #OUT_Message;
      JU    Z013;
// Stati di destinazione
Y013: L     16;
      T     #StatoSeguente;
Z013: NOP   0;
NETWORK
TITLE = State <16>: Blocca cassetto e prenota ribaditrice
      A     "Op40.Cycles".General.State.State_Bit[16];
      JCN   Z016;
      A     "Op40.Bench.MapE".Unlock_parts_down;
      A     "Op40.Bench.MapE".Box_index_down;
      A     "Op40.Bench.Systems".State.Cassetto_dentro;
      A     "Op40.Bench.Systems".State._Ribaditrice_a_disposiz;
      JC    Y016;
// Messaggi
// Blocco cassetto in corso
      AN    "Op40.Bench.MapE".Unlock_parts_down;
      ON    "Op40.Bench.MapE".Box_index_down;
      ON    "Op40.Bench.Systems".State.Cassetto_dentro;
      JC    A016;
// Attesa prenotazione ribaditrice
      AN    "Op40.Bench.Systems".State._Ribaditrice_a_disposiz;
      JC    B016;
      JU    B016;
A016: L     "Op40.Cycles".General.State.Page;
      T     #OUT_Page;
      L     8;	// Blocco cassetto in corso
      T     #OUT_Message;
      JU    Z016;
B016: L     "Op40.Cycles".General.State.Page;
      T     #OUT_Page;
      L     9;	//  Attesa prenotazione ribaditrice
      T     #OUT_Message;
      JU    Z016;
// Stati di destinazione
Y016: L     20;
      T     #StatoSeguente;
Z016: NOP   0;
NETWORK
TITLE = State <20>: Vai a quota di ribaditura punto corrente
      A     "Op40.Cycles".General.State.State_Bit[20];
      JCN   Z020;
      A     "Op40.Bench.Systems".State._Assi_posiz_raggiunta;
      A     "Op40.Bench.Systems".State.Ribaditrice_in_marcia;
      JC    Y020;
// Messaggi
// Posizionamento assi
      L     "Op40.Cycles".General.State.Page;
      T     #OUT_Page;
      L     15;	// Posizionamento assi
      T     #OUT_Message;
      JU    Z020;
// Stati di destinazione
Y020: L     25;
      T     #StatoSeguente;
Z020: NOP   0;
NETWORK
TITLE = State <25>: Esegui ribaditura punto corrente
      A     "Op40.Cycles".General.State.State_Bit[25];
      JCN   Z025;
      A     "Op40.Bench.Systems".State.Ribaditura_effettuata;
      JC    Y025;
// Messaggi
// Ribaditura spacer in corso
      L     "Op40.Cycles".General.State.Page;
      T     #OUT_Page;
      L     10;	// Ribaditura spacer in corso
      T     #OUT_Message;
      JU    Z025;
// Stati di destinazione
Y025: L     30;
      T     #StatoSeguente;
Z025: NOP   0;
NETWORK
TITLE = State <30>: Risali ribaditrice
      A     "Op40.Cycles".General.State.State_Bit[30];
      JCN   Z030;
      A     "Op40.Bench.Systems".State.Ribaditrice_alta;
      A(;
      L     "Op40.Bench.Systems".Data.Num_punto_in_lavorazione;
      L     "Op40.Bench.Recipe".NumeroPosizioni;
      <I;
      );
      JC    Y030;
      A     "Op40.Bench.Systems".State.Ribaditrice_alta;
      A(;
      L     "Op40.Bench.Systems".Data.Num_punto_in_lavorazione;
      L     "Op40.Bench.Recipe".NumeroPosizioni;
      >=I;
      );
      JC    X030;
// Messaggi
// Ribaditura spacer in corso
      L     "Op40.Cycles".General.State.Page;
      T     #OUT_Page;
      L     10;	// Ribaditura spacer in corso
      T     #OUT_Message;
      JU    Z030;
// Stati di destinazione
Y030: L     20;
      T     #StatoSeguente;
      JU    Z030;
X030: L     35;
      T     #StatoSeguente;
Z030: NOP   0;
NETWORK
TITLE = State <35>: Sblocco index e cassetto fuori
      A     "Op40.Cycles".General.State.State_Bit[35];
      A     "Op40.Bench.Systems".State.Cassetto_fuori;
      L     S5T#500MS;
      SD    "OP40St35_Cassetto_fuori";
      A     "Op40.Cycles".General.State.State_Bit[35];
      JCN   Z035;
      A     "Op40.Bench.MapE".Box_index_up;
      A     "OP40St35_Cassetto_fuori";
      JC    Y035;
// Messaggi
// Sblocco index in corso
      AN    "Op40.Bench.MapE".Box_index_up;
      JC    A035;
// Porta cassetto in zona di carico
      JU    B035;
A035: L     "Op40.Cycles".General.State.Page;
      T     #OUT_Page;
      L     11;	// Sblocco index in corso
      T     #OUT_Message;
      JU    Z035;
B035: L     "Op40.Cycles".General.State.Page;
      T     #OUT_Page;
      L     12;	// Porta cassetto in zona di carico
      T     #OUT_Message;
      JU    Z035;
// Stati di destinazione
Y035: L     40;
      T     #StatoSeguente;
Z035: NOP   0;
NETWORK
TITLE = State <40>: Sblocco pezzo e fine lavorazione
      A     "Op40.Cycles".General.State.State_Bit[40];
      JCN   Z040;
      A     "Op40.Bench.MapE".Box_index_down;
      A     "Op40.Bench.MapE".Unlock_parts_up;
      A     "Op40.Bench.Systems".State.Cassetto_fuori;
      A(;
      AN    "Op40.Tools.MapE".Presenza_pin_roller;
      O     "Op40.Bench.Recipe".Disable.CkPresenzaNozzleRing;
//     O     "Op40.Bench.Recipe".Disable.CkPresenzaPipe
      );
      JC    Y040;
// Messaggi
// Blocco index e sblocco pezzo in corso
      AN    "Op40.Bench.MapE".Box_index_down;
      ON    "Op40.Bench.MapE".Unlock_parts_up;
      JC    A040;
// Rimuovi pezzo buono dalla stazione
      JU    B040;
A040: L     "Op40.Cycles".General.State.Page;
      T     #OUT_Page;
      L     13;	// Blocco index e sblocco pezzo in corso
      T     #OUT_Message;
      JU    Z040;
B040: L     "Op40.Cycles".General.State.Page;
      T     #OUT_Page;
      L     14;	// Rimuovi pezzo buono dalla stazione
      T     #OUT_Message;
      JU    Z040;
// Stati di destinazione
Y040: L     60;
      T     #StatoSeguente;
Z040: NOP   0;
NETWORK
TITLE =
      A     "Op40.Cycles".General.State.State_Bit[60];
      JCN   Z060;
// Stati di destinazione
      L     10;
      T     #StatoSeguente;
Z060: NOP   0;
NETWORK
TITLE = Output
      L     #Stato;
      T     #OUT_CicloStato;
      A     #Stat_CicloInCorso;
      =     #OUT_St_CicloInCorso;
      A     #Stat_CicloTermOk;
      =     #OUT_St_CicloTerminatoOK;
      A     #Stat_CicloTermKO;
      =     #OUT_St_CicloTerminatoKO;
END_FUNCTION_BLOCK

FUNCTION_BLOCK "Op40.Cycle.Restore"	// FB 221
VERSION : 0.1
VAR_INPUT
  IN_Cm_ON : BOOL ;	//1: Attiva il ciclo; 0: Reset del ciclo
  IN_HOLD : BOOL ;	//Blocca il ciclo nel passo successivo
  IN_STEP : BOOL ;
END_VAR
VAR_OUTPUT
  OUT_St_CicloInCorso : BOOL ;
  OUT_St_CicloTerminatoOK : BOOL ;
  OUT_St_CicloTerminatoKO : BOOL ;
  OUT_CicloStato : INT ;
  OUT_Page : INT ;
  OUT_Message : INT ;
END_VAR
VAR
  Stato : INT ;
  StatoSeguente : INT ;
  FrontePassoSingolo : BOOL ;
  Stat_CicloTermOk : BOOL ;
  Stat_CicloTermKO : BOOL ;
  Stat_CicloInCorso : BOOL ;
  Timer_Pennarello : SFB 4;
END_VAR
VAR_TEMP
  Pag_Active : ARRAY  [0 .. 100 ] OF BOOL ;
END_VAR
BEGIN
NETWORK
TITLE = FLOW CHART
NETWORK
TITLE = Update state
      A     #IN_Cm_ON;
      JC    M002;
      L     0;
      T     #Stato;
      T     #StatoSeguente;
M002: NOP   0;
//->Update State
      A     #IN_STEP;
      FP    #FrontePassoSingolo;
      ON    #IN_HOLD;	//se usassi UN l'Hold agirebbe anche su avanzamento a passo singolo 
      JCN   N100;
      L     #StatoSeguente;
      T     #Stato;
N100: NOP   0;
// determinazione bit di stato
      CALL  "Conv_INT->BIT" (
           Valore                   := #Stato,
           States                   := "Op40.Cycles".Restore.State.State_Bit);
NETWORK
TITLE = Detect page active from OP
// serve??????
//      CALL  "Conv_INT->BIT"
//       Valore:=DB325.DBW2
//       States:=#Pag_Active
NETWORK
TITLE = States particular
      L     #Stato;
      L     0;
      <>I;
//->Evita ritardi
      A     #IN_Cm_ON;
      =     #Stat_CicloInCorso;
      A     "Op40.Cycles".Restore.State.State_Bit[60];
      =     #Stat_CicloTermOk;
      A     "Op40.Cycles".Restore.State.State_Bit[63];
      =     #Stat_CicloTermKO;
NETWORK
TITLE = Diagnostic default
//    L     0
//    T     #Page
//    L     0
//    T     #Message 
//      L     6
//      T     #StatoSeguente
NETWORK
TITLE = State <0>: Ciclo off
      A     "Op40.Cycles".Restore.State.State_Bit[0];
      A     #IN_Cm_ON;
      JC    A000;
      L     "Op10.Cycles".Restore.State.Page;
      T     #OUT_Page;
      L     20;	// ciclo off
      T     #OUT_Message;
      JU    Z000;
A000: L     10;
      T     #StatoSeguente;
Z000: NOP   0;
NETWORK
TITLE = State <10>: Sali ribaditrice
      A     "Op40.Cycles".Restore.State.State_Bit[10];
      JCN   Z010;
      A     "Op40.Bench.Systems".State.Ribaditrice_alta;
      O     "Op40.Bench.Systems".State._Ribad_in_fuori_ingombro;
      AN    "Op40.Bench.MapE".Box_out;
      JC    Y010;
      A     "Op40.Bench.Systems".State.Ribaditrice_alta;
      O     "Op40.Bench.Systems".State._Ribad_in_fuori_ingombro;
      A     "Op40.Bench.MapE".Box_out;
      JC    X010;
// Messaggi
// Salita ribaditrice in corso
//      UN    "Op40.Bench.Systems".State.Ribaditrice_alta
//      UN    DB205.DBX    11.7
//      SPA   A010
      L     "Op40.Cycles".Restore.State.Page;
      T     #OUT_Page;
      L     21;	// Salita ribaditrice in corso
      T     #OUT_Message;
      JU    Z010;
// Stati di destinazione
Y010: L     15;
      T     #StatoSeguente;
      JU    Z010;
X010: L     20;
      T     #StatoSeguente;
Z010: NOP   0;
NETWORK
TITLE = State <15>: Sblocca index e cassetto fuori
      A     "Op40.Cycles".Restore.State.State_Bit[15];
      A     "Op40.Bench.Systems".State.Cassetto_fuori;
      L     S5T#500MS;
      SD    "RS40St15_Cassetto_fuori";
      A     "Op40.Cycles".Restore.State.State_Bit[15];
      JCN   Z015;
      A     "Op40.Bench.MapE".Box_index_up;
      A     "RS40St15_Cassetto_fuori";
      JC    Y015;
// Messaggi
//   Sblocco index in corso
      AN    "Op40.Bench.MapE".Box_index_up;
      JC    A015;
// Porta cassetto in zona di scarico
      JU    B015;
A015: L     "Op40.Cycles".Restore.State.Page;
      T     #OUT_Page;
      L     22;	//  Sblocco index in corso
      T     #OUT_Message;
      JU    Z015;
B015: L     "Op40.Cycles".Restore.State.Page;
      T     #OUT_Page;
      L     23;	// Porta cassetto in zona di scarico
      T     #OUT_Message;
      JU    Z015;
// Stati di destinazione
Y015: L     20;
      T     #StatoSeguente;
Z015: NOP   0;
NETWORK
TITLE = State <20>: Blocca index e sblocca pezzo - rimuovi scarto
      A     "Op40.Cycles".Restore.State.State_Bit[20];
      JCN   Z020;
      A     "Op40.Bench.MapE".Unlock_parts_up;
      A     "Op40.Bench.MapE".Box_index_down;
      A     "Op40.Bench.Systems".State.Cassetto_fuori;
      A(;
      AN    "Op40.Tools.MapE".Presenza_pin_roller;
      O     "Op40.Bench.Recipe".Disable.CkPresenzaNozzleRing;	//MDQ
//      O     "Op40.Bench.Recipe".Disable.CkPresenzaPipe
      );
      JC    Y020;
// Messaggi
// Blocco index e sblocco pezzo in corso
      AN    "Op40.Bench.MapE".Unlock_parts_up;
      ON    "Op40.Bench.MapE".Box_index_down;
      ON    "Op40.Bench.Systems".State.Cassetto_fuori;
      JC    A020;
// Rimuovi pezzo scarto dalla stazione
      JU    B020;
A020: L     "Op40.Cycles".Restore.State.Page;
      T     #OUT_Page;
      L     24;	// Blocco index e sblocco pezzo in corso
      T     #OUT_Message;
      JU    Z020;
B020: L     "Op40.Cycles".Restore.State.Page;
      T     #OUT_Page;
      L     25;	// Rimuovi pezzo scarto dalla stazione
      T     #OUT_Message;
      JU    Z020;
// Stati di destinazione
Y020: L     60;
      T     #StatoSeguente;
Z020: NOP   0;
NETWORK
TITLE = Output
      L     #Stato;
      T     #OUT_CicloStato;
      A     #Stat_CicloInCorso;
      =     #OUT_St_CicloInCorso;
      A     #Stat_CicloTermOk;
      =     #OUT_St_CicloTerminatoOK;
      A     #Stat_CicloTermKO;
      =     #OUT_St_CicloTerminatoKO;
END_FUNCTION_BLOCK

FUNCTION_BLOCK "Std_Sinamics_Axis"	// FB 450
//Gestione di sistema di max 4 assi (X-Y-Z-U) mediante SIEMENS SINAMICS CU320 
//
AUTHOR : Castel
VERSION : 0.1
VAR_INPUT
  Enable_Function : BOOL ;	//Abilitazione esecuzione blocco
  AddrIN : WORD ;
  AddrOUT : WORD ;
  Cmd_Jog_Minus_Axis : BOOL ;	//Start movimento incrementale negativa asse
  Cmd_Jog_Plus_Axis : BOOL ;	//Start movimento incrementale positiva asse
  Cmd_Start_Posit_Axis : BOOL ;	//Muovi alla posizione programmata asse
  Cmd_Reference_Axis : BOOL ;	//Ricerca punto di riferimento
  In_Reference_Cam : BOOL ;	//Camma punto di riferimento
  Cmd_Enable_Axis : BOOL ;	//Abbilita la regolazione rampa
  Cmd_ResetAlarm : BOOL ;	//Reset Allarmi
  Cmd_Override_Axis : INT ;	//Valore override 0..100% asse
  Cmd_Acceleration_Axis : INT ;	//Valore accellerazione 0..100% asse
  Cmd_Deceleration_Axis : INT ;	//Valore decellerazione 0..100% asse
  Cmd_Speed_Axis : DINT ;	//Valore velocita asse
  Cmd_Position_Axis : DINT ;	//Posizione assoluta da raggiungere in micron asse
  Cmd_Positioning_Mode : INT ;	//0=Assoluto, 1=relativo, 2=AssolutoPiu, 3 AssolutoMeno
END_VAR
VAR_OUTPUT
  Profibus_Write_Error : BOOL ;	//Errore nella scrittura dati nella rete Profibus
  Profibus_Read_Error : BOOL ;	//Errore nella lettura dati dalla rete Profibus
  St_Referenced_Axis : BOOL ;	//Arre referenziato
  St_Pos_Axis_OK : BOOL ;	//Posizione asse raggiunta
  St_Axis_Running : BOOL ;	//Asse in movimento
  St_Alarm_Code_Axis : BYTE ;	//Rispote d'errore in codice dall'asse
  St_Position_Axis : DINT ;	//Posizione assoluta asse in micron
  St_EndstrokePlus_Reached : BOOL ;
  St_EndstrokeMinu_Reached : BOOL ;
  St_Axis_ReadyToStart : BOOL ;
END_VAR
VAR
  Asse_ERR_Ricezione : BOOL ;
  Asse_ERR_Trasmissione : BOOL ;
  AsseMossoInPosizioname : BOOL ;
  Axis_Buffer : UDT 450;
END_VAR
VAR_TEMP
  RET_VAL_Write_Axis : INT ;	//Valore di ritorno per diagnosi SFC
  RET_VAL_Read_Axis : INT ;	//Valore di ritorno per diagnosi SFC
  Override_Axis : INT ;
  Acceleration_Axis : INT ;
  Deceleration_Axis : INT ;
  Speed_Axis : DINT ;
END_VAR
BEGIN
NETWORK
TITLE =
      A     #Enable_Function;
      JCN   m000;
NETWORK
TITLE = Lettura dati SINAMICS ASSE X
//Utilizzato Telegramma SIEMENS 110, PZD-12/7
      CALL  "DPRD_DAT" (
           LADDR                    := #AddrIN,
           RET_VAL                  := #RET_VAL_Read_Axis,
           RECORD                   := #Axis_Buffer.IN);	// Byte 310       // Indirizzo iniziale di lettura dalla config. Hw convertito in Hex. / #P_Buffer               //P#DB141.DBX0.0 BYTE 14
NETWORK
TITLE = Anomalia ricezione dati SINAMICS ASSE X
      A(;
      L     #RET_VAL_Read_Axis;
      L     W#16#8000;
      >=I;
      );
      A(;
      L     #RET_VAL_Read_Axis;
      L     W#16#8FFF;
      <=I;
      );
      =     #Asse_ERR_Ricezione;
NETWORK
TITLE =
//***************************** ASSE X **************************************
NETWORK
TITLE = Override asse X
//Campo di lavoro del parametro accellerazione 0..100%
      L     #Cmd_Override_Axis;
      T     #Override_Axis;
      L     #Override_Axis;
      L     100;
      >I;
      JCN   m010;
      L     100;
      T     #Override_Axis;
m010: NOP   0;
      L     #Override_Axis;
      L     0;
      <I;
      JCN   m011;
      L     0;
      T     #Override_Axis;
m011: NOP   0;
      L     #Override_Axis;	// VALORE 0-100% OVERRIDE VALORE DI COMANDO
      ITD;
      L     L#32767;
      *D;
      L     L#100;
      /D;
      T     #Axis_Buffer.OUT.OUT_PZD5;	//  "Telegramma Asse X".OUT.OUT_PZD5    // override max  0..32767    
NETWORK
TITLE = MDI Accelerazione asse X
//Campo di lavoro del parametro accellerazione 0..100%
      L     #Cmd_Acceleration_Axis;
      T     #Acceleration_Axis;
      L     #Acceleration_Axis;
      L     100;
      >I;
      JCN   m020;
      L     100;
      T     #Acceleration_Axis;
m020: NOP   0;
      L     #Acceleration_Axis;
      L     0;
      <I;
      JCN   m021;
      L     0;
      T     #Acceleration_Axis;
m021: NOP   0;
      L     #Acceleration_Axis;	//VALORE 0-100% ACCELERAZIONE VALORE DI COMANDO
      ITD;
      L     L#32767;
      *D;
      L     L#100;
      /D;
      T     #Axis_Buffer.OUT.OUT_PZD10;	//  "Telegramma Asse X".OUT.OUT_PZD10    // MDI accelerazione max  0..32767  
NETWORK
TITLE = MDI Decelerazione asse X
//Campo di lavoro del parametro accellerazione 0..100%
      L     #Cmd_Deceleration_Axis;
      T     #Deceleration_Axis;
      L     #Deceleration_Axis;
      L     100;
      >I;
      JCN   m030;
      L     100;
      T     #Deceleration_Axis;
m030: NOP   0;
      L     #Deceleration_Axis;
      L     0;
      <I;
      JCN   m031;
      L     0;
      T     #Deceleration_Axis;
m031: NOP   0;
      L     #Deceleration_Axis;	//VALORE 0-100% DECELERAZIONE VALORE DI COMANDO
      ITD;
      L     L#32767;
      *D;
      L     L#100;
      /D;
      T     #Axis_Buffer.OUT.OUT_PZD11;	// "Telegramma Asse X".OUT.OUT_PZD11    // MDI decelerazione max  0..32767  
NETWORK
TITLE = MDI Velocità asse X
//Campo di lavoro del parametro decellerazione 0..100%
      L     #Cmd_Speed_Axis;
      T     #Speed_Axis;
      L     #Speed_Axis;
      L     L#30000;
      >D;
      JCN   m040;
      L     L#30000;
      T     #Speed_Axis;
m040: NOP   0;
      L     #Speed_Axis;
      L     L#0;
      <D;
      JCN   m041;
      L     L#0;
      T     #Speed_Axis;
m041: NOP   0;
      L     #Speed_Axis;	//VALORE 0-100% VELOCITA' VALORE DI COMANDO
      T     #Axis_Buffer.OUT.OUT_PZD8_9;	// "Telegramma Asse X".OUT.OUT_PZD8_9    // MDI velocità max  0..30000 
NETWORK
TITLE = MDI Posizione da raggiungere asse X
      L     #Cmd_Position_Axis;
      T     #Axis_Buffer.OUT.OUT_PZD6_7;	// "Telegramma Asse X".OUT.OUT_PZD6_7    // Posizione assoluta da raggiungere un micron
NETWORK
TITLE = MDI Mode asse (Assoluto o Relativo)
//xx0x hex -> assoluto
//xx1x hex -> relativo
//xx2x hex -> ass_pos (solo per correzione modulo)
//xx3x hex -> ass_neg (solo per correzione modulo)
//
// Default posizionamento assoluto!!!
      L     #Cmd_Positioning_Mode;
      JL    Mox;
      JU    Mo0;
      JU    Mo1;
      JU    Mo2;
      JU    Mo3;
Mox:  JU    Mo0;
Mo0:  L     0;	// Posizionamento assoluto
      JU    MoR;
Mo1:  L     W#16#10;	// Posizionamento relativo
      JU    MoR;
Mo2:  L     W#16#20;	// Posizionamento assoluto Più (con modulo)
      JU    MoR;
Mo3:  L     W#16#30;	// Posizionamento assoluto Meno (con modulo)
      JU    MoR;
MoR:  T     #Axis_Buffer.OUT.OUT_PZD12;
NETWORK
TITLE = PACO1 gestione parola di comando 1 asse X
//
//
//
//
// PACO1 Bit10 controllo da plc (abilitazione profibus)
      SET;
      =     #Axis_Buffer.OUT.OUT_PZD1_BIT10;	// conduzione profibus    
      =     #Axis_Buffer.OUT.OUT_PZD1_BIT5;	// NO Arresto immediato
      =     #Axis_Buffer.OUT.OUT_PZD2_BIT15;	// abilita rampa 
// Reset alarm
      A     #Cmd_ResetAlarm;
      =     #Axis_Buffer.OUT.OUT_PZD1_BIT7;	// "Telegramma Asse X".OUT.OUT_PZD1_BIT7
// Abilitazione asse
      A     #Cmd_Enable_Axis;
      =     #Axis_Buffer.OUT.OUT_PZD1_BIT1;
      =     #Axis_Buffer.OUT.OUT_PZD1_BIT2;
      =     #Axis_Buffer.OUT.OUT_PZD1_BIT3;	// "Telegramma Asse X".OUT.OUT_PZD1_BIT3    // Abilita al funzionamento 
      A     #Cmd_Enable_Axis;
      A     #Axis_Buffer.IN.IN_PZD1_BIT4;
      A     #Axis_Buffer.IN.IN_PZD1_BIT5;
      A     #Axis_Buffer.IN.IN_PZD1_BIT0;
      S     #Axis_Buffer.OUT.OUT_PZD1_BIT0;
      AN    #Cmd_Enable_Axis;
      R     #Axis_Buffer.OUT.OUT_PZD1_BIT0;
// Marcia a impulsi jog negativo asse
      A     #Cmd_Jog_Minus_Axis;
      AN    #Cmd_Jog_Plus_Axis;
      AN    #Cmd_Reference_Axis;
      AN    #Cmd_Start_Posit_Axis;
      =     #Axis_Buffer.OUT.OUT_PZD1_BIT8;	// jog negativo        
// Marcia a impulsi jog positivo asse
      AN    #Cmd_Jog_Minus_Axis;
      A     #Cmd_Jog_Plus_Axis;
      AN    #Cmd_Reference_Axis;
      AN    #Cmd_Start_Posit_Axis;
      =     #Axis_Buffer.OUT.OUT_PZD1_BIT9;	// jog positivo     
// Ricerca punto di zero
      A     #Cmd_Reference_Axis;
      AN    #Cmd_Jog_Minus_Axis;
      AN    #Cmd_Jog_Plus_Axis;
      AN    #Cmd_Start_Posit_Axis;
      =     #Axis_Buffer.OUT.OUT_PZD1_BIT11;	// avvio del punto di riferimento  (ricerca zero)
// Camma punto di zero
      A     #In_Reference_Cam;
      =     #Axis_Buffer.OUT.OUT_PZD3_BIT2;	// Camma di zero
// Comando di marcia
      A     #Axis_Buffer.OUT.OUT_PZD1_BIT0;	// OFF-1 
      A     #Axis_Buffer.OUT.OUT_PZD1_BIT1;	// OFF-2
      A     #Axis_Buffer.OUT.OUT_PZD1_BIT2;	// OFF-3   
      A     #Axis_Buffer.IN.IN_PZD1_BIT0;
      A     #Axis_Buffer.IN.IN_PZD1_BIT1;
      A     #Axis_Buffer.IN.IN_PZD1_BIT2;
      AN    #Axis_Buffer.IN.IN_PZD1_BIT3;
      A     #Axis_Buffer.IN.IN_PZD1_BIT4;
      A     #Axis_Buffer.IN.IN_PZD1_BIT5;
      AN    #Axis_Buffer.IN.IN_PZD1_BIT6;
      AN    #Cmd_Reference_Axis;
      AN    #Cmd_Jog_Minus_Axis;
      AN    #Cmd_Jog_Plus_Axis;
      A     #Cmd_Start_Posit_Axis;
      =     #Axis_Buffer.OUT.OUT_PZD1_BIT6;	// Attiva movimento
      =     #Axis_Buffer.OUT.OUT_PZD1_BIT4;	// Rifiuto job di movimento
NETWORK
TITLE = Posizione reale assoluta dell'asse X
      L     #Axis_Buffer.IN.IN_PZD6_7;	// "Telegramma Asse X".IN.IN_PZD6_7
      T     #St_Position_Axis;
NETWORK
TITLE = Posizione richiesta raggiunta asse X
// Registra movimento avvenuto asse in posizioamento
      AN    #Axis_Buffer.IN.IN_PZD1_BIT10;
      ON    #Axis_Buffer.IN.IN_PZD1_BIT13;
      A     #Cmd_Start_Posit_Axis;
      S     #AsseMossoInPosizioname;
      AN    #Cmd_Start_Posit_Axis;
      R     #AsseMossoInPosizioname;
      L     #Cmd_Positioning_Mode;
      L     1;
      ==I;
      JC    NABS;
// Controlo posizione raggiunta se posizionamento assoluto
      A(;
      L     #Axis_Buffer.IN.IN_PZD6_7;	// "Telegramma Asse X".IN.IN_PZD6_7
      L     L#200;
      +D;
      L     #Axis_Buffer.OUT.OUT_PZD6_7;	// "Telegramma Asse X".OUT.OUT_PZD6_7
      >=D;
      );
      A(;
      L     #Axis_Buffer.IN.IN_PZD6_7;	// "Telegramma Asse X".IN.IN_PZD6_7
      L     L#200;
      -D;
      L     #Axis_Buffer.OUT.OUT_PZD6_7;	// "Telegramma Asse X".OUT.OUT_PZD6_7
      <=D;
      );
      A     #Axis_Buffer.IN.IN_PZD1_BIT10;
      A     #Axis_Buffer.IN.IN_PZD1_BIT13;
      A     #Cmd_Start_Posit_Axis;
      =     #St_Pos_Axis_OK;
      JU    FPOK;
NABS: NOP   0;
// Controlo posizione raggiunta se posizionamento relativo
      A     #Axis_Buffer.IN.IN_PZD1_BIT10;
      A     #Axis_Buffer.IN.IN_PZD1_BIT13;
      A     #Cmd_Start_Posit_Axis;
      A     #AsseMossoInPosizioname;
      =     #St_Pos_Axis_OK;
FPOK: NOP   0;
NETWORK
TITLE = Asse X in movimento dopo lo start al Job
      A     #Axis_Buffer.IN.IN_PZD3_BIT4;
      O     #Axis_Buffer.IN.IN_PZD3_BIT5;
      =     #St_Axis_Running;
NETWORK
TITLE = Asse referenziato
      A     #Axis_Buffer.IN.IN_PZD1_BIT11;
      =     #St_Referenced_Axis;
NETWORK
TITLE = Segnalazioni errori o anomalie asse X
      A     #Axis_Buffer.IN.IN_PZD1_BIT3;	//  "Telegramma Asse X".IN.IN_PZD1_BIT3
      JC    m063;
      AN    #Axis_Buffer.IN.IN_PZD1_BIT0;	// "Telegramma Asse X".IN.IN_PZD1_BIT0
      JC    m060;
      AN    #Axis_Buffer.IN.IN_PZD1_BIT1;	// "Telegramma Asse X".IN.IN_PZD1_BIT1
      JC    m061;
      AN    #Axis_Buffer.IN.IN_PZD1_BIT2;	// "Telegramma Asse X".IN.IN_PZD1_BIT2
      JC    m062;
      AN    #Axis_Buffer.IN.IN_PZD1_BIT4;	// "Telegramma Asse X".IN.IN_PZD1_BIT4
      JC    m064;
      AN    #Axis_Buffer.IN.IN_PZD1_BIT5;	// "Telegramma Asse X".IN.IN_PZD1_BIT5
      JC    m065;
      A     #Axis_Buffer.IN.IN_PZD1_BIT6;	// "Telegramma Asse X".IN.IN_PZD1_BIT6
      JC    m066;
      A     #Axis_Buffer.IN.IN_PZD3_BIT6;	// "Telegramma Asse X".IN.IN_PZD3_BIT6
      JC    m067;
      A     #Axis_Buffer.IN.IN_PZD3_BIT7;	// "Telegramma Asse X".IN.IN_PZD3_BIT7
      JC    m068;
      JU    m070;
m060: L     1;	// Cod.1: asse non pronto all'inserzione
      JU    m079;
m061: L     2;	// Cod.2: asse non pronto al funzionamento
      JU    m079;
m062: L     3;	// Cod.3: asse non abilitato
      JU    m079;
m063: L     4;	// Cod.4: asse in anomalia
      JU    m079;
m064: L     5;	// Cod.5: asse in arresto per inerzia  (OFF-2)
      JU    m079;
m065: L     6;	// Cod.6: asse in arresto rapido (OFF-3)
      JU    m079;
m066: L     7;	// Cod.7: blocco all'inserzione dell'asse
      JU    m079;
m067: L     8;	// Cod.8: finecorsa SW- raggiunto
      JU    m079;
m068: L     9;	// Cod.9: finecorsa SW+ raggiunto
      JU    m079;
m070: L     0;	// Nessun errore dall'asse
      JU    m079;
m079: T     #St_Alarm_Code_Axis;
NETWORK
TITLE = Invio dati SINAMICS ASSE X
//Utilizzato Telegramma SIEMENS 110, PZD-12/7
      CALL  "DPWR_DAT" (
           LADDR                    := #AddrOUT,
           RECORD                   := #Axis_Buffer.OUT,
           RET_VAL                  := #RET_VAL_Write_Axis);	//Byte 352       // Indirizzo iniziale di scrittura dalla config. Hw convertito in Hex.
NETWORK
TITLE = Anomalia invio dati SINAMICS ASSE X
      A(;
      L     #RET_VAL_Write_Axis;
      L     W#16#8000;
      >=I;
      );
      A(;
      L     #RET_VAL_Write_Axis;
      L     W#16#8FFF;
      <=I;
      );
      =     #Asse_ERR_Trasmissione;
      NOP   0;
NETWORK
TITLE = Segnalazioni errore profibus
      A     #Asse_ERR_Trasmissione;
      =     #Profibus_Write_Error;
      A     #Asse_ERR_Ricezione;
      =     #Profibus_Read_Error;
NETWORK
TITLE =
      A     #Axis_Buffer.IN.IN_PZD3_BIT7;
      =     #St_EndstrokePlus_Reached;
      A     #Axis_Buffer.IN.IN_PZD3_BIT6;
      =     #St_EndstrokeMinu_Reached;
      A     #Axis_Buffer.IN.IN_PZD1_BIT0;
      A     #Axis_Buffer.IN.IN_PZD1_BIT1;
      A     #Axis_Buffer.IN.IN_PZD1_BIT2;
      A     #Axis_Buffer.IN.IN_PZD1_BIT8;
      A     #Axis_Buffer.IN.IN_PZD1_BIT11;
      =     #St_Axis_ReadyToStart;
NETWORK
TITLE =
m000: NOP   0;
END_FUNCTION_BLOCK

FUNCTION_BLOCK "Std.Sinamics_Cu_S"	// FB 455
//Gestione di sistema assi mediante SIEMENS SINAMICS CU320 
//
VERSION : 0.1
VAR_INPUT
  IN_Enable : BOOL ;	//Abilitazione esecuzione blocco
  IN_Addr_Read : WORD ;	//Indirizzo iniziale di lettura dati da profibus in cod. esadecimale
  IN_Addr_Write : WORD ;	//Indirizzo iniziale di scrittura dati nel profibus in cod. esadecimale
END_VAR
VAR_OUTPUT
  OUT_HW_DI0 : BOOL ;
  OUT_HW_DI1 : BOOL ;
  OUT_HW_DI2 : BOOL ;
  OUT_HW_DI3 : BOOL ;
  OUT_HW_DI4 : BOOL ;
  OUT_HW_DI5 : BOOL ;
  OUT_HW_DI6 : BOOL ;
  OUT_HW_DI7 : BOOL ;
  OUT_HW_DI8 : BOOL ;
  OUT_HW_DI9 : BOOL ;
  OUT_HW_DI10 : BOOL ;
  OUT_HW_DI11 : BOOL ;
  OUT_HW_DI12 : BOOL ;
  OUT_HW_DI13 : BOOL ;
  OUT_HW_DI14 : BOOL ;
  OUT_HW_DI15 : BOOL ;
  OUT_Profibus_Write_Error : BOOL ;	//Errore nella scrittura dati nella rete Profibus
  OUT_Profibus_Read_Error : BOOL ;	//Errore nella lettura dati dalla rete Profibus
END_VAR
VAR
  CU320_ERR_Ricezione : BOOL ;
  CU320_ERR_Trasmissione : BOOL ;
  Cu320_Buffer : UDT 455;
END_VAR
VAR_TEMP
  Dummy : BOOL ;
  RET_VAL_Write_CU320 : INT ;	//Valore di ritorno per diagnosi SFC
  RET_VAL_Read_CU320 : INT ;	//Valore di ritorno per diagnosi SFC
END_VAR
BEGIN
NETWORK
TITLE =
      AN    #IN_Enable;
      R     #OUT_Profibus_Write_Error;
      R     #OUT_Profibus_Read_Error;
      JC    m000;
NETWORK
TITLE = Lettura dati SINAMICS Control unit CU320
//Utilizzato Telegramma SIEMENS 390, PZD-2/2
      CALL  "DPRD_DAT" (
           LADDR                    := #IN_Addr_Read,
           RET_VAL                  := #RET_VAL_Read_CU320,
           RECORD                   := #Cu320_Buffer.IN);
NETWORK
TITLE = Anomalia ricezione dati SINAMICS Cu320
      A(;
      L     #RET_VAL_Read_CU320;
      L     W#16#8000;
      >=I;
      );
      A(;
      L     #RET_VAL_Read_CU320;
      L     W#16#8FFF;
      <=I;
      );
      =     #CU320_ERR_Ricezione;
NETWORK
TITLE = Parole di stato telegramma Cu320
// Segnale di richiesta reset Sinamics dall'esterno
      A     #Cu320_Buffer.IN.IN_PZD2_BIT0;
      =     #OUT_HW_DI8;
      A     #Cu320_Buffer.IN.IN_PZD2_BIT1;
      =     #OUT_HW_DI9;
      A     #Cu320_Buffer.IN.IN_PZD2_BIT2;
      =     #OUT_HW_DI10;
      A     #Cu320_Buffer.IN.IN_PZD2_BIT3;
      =     #OUT_HW_DI11;
      A     #Cu320_Buffer.IN.IN_PZD2_BIT4;
      =     #OUT_HW_DI12;
      A     #Cu320_Buffer.IN.IN_PZD2_BIT5;
      =     #OUT_HW_DI13;
      A     #Cu320_Buffer.IN.IN_PZD2_BIT6;
      =     #OUT_HW_DI14;
      A     #Cu320_Buffer.IN.IN_PZD2_BIT7;
      =     #OUT_HW_DI15;
      A     #Cu320_Buffer.IN.IN_PZD2_BIT8;
      =     #OUT_HW_DI0;
      A     #Cu320_Buffer.IN.IN_PZD2_BIT9;
      =     #OUT_HW_DI1;
      A     #Cu320_Buffer.IN.IN_PZD2_BIT10;
      =     #OUT_HW_DI2;
      A     #Cu320_Buffer.IN.IN_PZD2_BIT11;
      =     #OUT_HW_DI3;
      A     #Cu320_Buffer.IN.IN_PZD2_BIT12;
      =     #OUT_HW_DI4;
      A     #Cu320_Buffer.IN.IN_PZD2_BIT13;
      =     #OUT_HW_DI5;
      A     #Cu320_Buffer.IN.IN_PZD2_BIT14;
      =     #OUT_HW_DI6;
      A     #Cu320_Buffer.IN.IN_PZD2_BIT15;
      =     #OUT_HW_DI7;
NETWORK
TITLE = Segnalazioni errore profibus
//      U     #CU320_ERR_Trasmissione
//      =     #OUT_Profibus_Write_Error
      A     #CU320_ERR_Ricezione;
      =     #OUT_Profibus_Read_Error;
      JU    m001;
m000: CLR;
      =     #OUT_HW_DI0;
      =     #OUT_HW_DI1;
      =     #OUT_HW_DI2;
      =     #OUT_HW_DI3;
      =     #OUT_HW_DI7;
      =     #OUT_HW_DI6;
      =     #OUT_HW_DI5;
      =     #OUT_HW_DI4;
      =     #OUT_HW_DI13;
      =     #OUT_HW_DI14;
      =     #OUT_HW_DI15;
      =     #OUT_HW_DI14;
m001: NOP   0;
NETWORK
TITLE = Azzera uscite con blocco disabilitato
END_FUNCTION_BLOCK

// FC 5: know-how protected block, not included

FUNCTION "Conv_INT->BIT" : VOID	// FC 17
AUTHOR : Filip1
NAME : StateBit
VERSION : 1.0
VAR_INPUT
  Valore : INT ;
END_VAR
VAR_IN_OUT
  States : ANY ;
END_VAR
VAR_TEMP
  CONTATORE : WORD ;
  Num_DB : INT ;
  Punt : DWORD ;
  Num_Bit : WORD ;
  Data_T : BYTE ;
  Punt_1 : DWORD ;
END_VAR
BEGIN
NETWORK
TITLE = Decodifica INT -> serie di bit
      L     P##States;
      LAR1;
      L     B [AR1,P#1.0];
      T     #Data_T;
      L     W [AR1,P#2.0];
      T     #Num_Bit;
      L     W [AR1,P#4.0];
      T     #Num_DB;
      L     D [AR1,P#6.0];
      T     #Punt;
      L     #Data_T;
      L     1;	//tipo di dati = 1 -> bool
      ==I;
      JC    OK;
      L     #Data_T;
      L     3;	//tipo di dati = 2 o 3 -> byte o char
      >I;
      JC    no_b;
      L     #Num_Bit;
      L     8;
      *I;
      T     #Num_Bit;
      JC    OK;
no_b: L     #Data_T;
      L     5;	//tipo di dati = 4 o 5 -> int o word
      >I;
      JC    Exit;
      L     #Num_Bit;
      L     16;
      *I;
      T     #Num_Bit;
      JC    OK;
      JCN   Exit;
OK:   OPN   DB [#Num_DB];
      L     #Punt;
      T     #Punt_1;
//- AZZERAMENTO INIZIALE
      L     #Num_Bit;
ZERO: T     #CONTATORE;
      L     #Punt_1;
      LAR1;
      SET;
      R      [AR1,P#0.0];
      L     #Punt_1;
      L     1;
      +D;
      T     #Punt_1;
      L     #CONTATORE;
      LOOP  ZERO;
//- LETTURA BIT DA SETTARE
      L     #Valore;
      L     #Num_Bit;
      <I;
      JCN   Exit;
      L     #Valore;
      L     #Punt;
      +D;
      LAR1;
      SET;
      S      [AR1,P#0.0];
Exit: NOP   0;
END_FUNCTION

FUNCTION "Bench.Mode" : VOID	// FC 20
VERSION : 0.1
VAR_INPUT
  Enable : BOOL ;	//Abilita le uscite: sempre a True
  AllarmeEmergenza : BOOL ;	//Presenza allarme di emergenza: se false -> Uscita PlcOk a 0
  AusiliariOK : BOOL ;	//Segnale Ausiliari pronto: per passaggio da modo Emergenza a modo Test Macchina
  ComandoTestMacchina : BOOL ;	//Segnale che forza il modo test Macchina (es. Pulsante di test lampade)
  ComandoSetup : BOOL ;	//Segnale che forza il modo Setuo (es. Selettore di setup)
  ComandoManuale : BOOL ;	//Interruttore con cui si desidera selezionare la modalità manuale
  ComandoAutomatico : BOOL ;	//Interruttore con cui si desidera selezionare la modalità automatica
  TimerTest : TIMER ;	//Timer per test dopo inserzione ausiliari
END_VAR
VAR_OUTPUT
  ModoEmergenza : BOOL ;
  ModoTestMacchina : BOOL ;
  ModoSetup : BOOL ;
  ModoManuale : BOOL ;
  ModoAutomatico : BOOL ;
  DO_PlcOk : BOOL ;
END_VAR
BEGIN
NETWORK
TITLE = Gestioni Modi
NETWORK
TITLE = MacchinaSpenta
      A     #Enable;
      JC    Enbl;
      R     #ModoEmergenza;
      R     #ModoTestMacchina;
      R     #ModoSetup;
      R     #ModoManuale;
      R     #ModoAutomatico;
      R     #DO_PlcOk;
      BEU;
Enbl: NOP   0;
NETWORK
TITLE = CASE Command
      A     #AusiliariOK;
      AN    #AllarmeEmergenza;
      L     S5T#2S;
      SD    #TimerTest;
      AN    #AusiliariOK;
      O     #AllarmeEmergenza;
      JC    Emer;
      A     #AusiliariOK;
      AN    #TimerTest;
      JC    Test;
      A     #TimerTest;
      A     #ComandoSetup;
      JC    Setu;
      A     #TimerTest;
      A(;
      A     #ComandoManuale;
      O     #ModoManuale;
      );
      AN    #ComandoAutomatico;
      JC    Manu;
      A     #TimerTest;
      A(;
      A     #ComandoAutomatico;
      O     #ModoAutomatico;
      );
      AN    #ComandoManuale;
      JC    Auto;
      JU    Setu;
NETWORK
TITLE = CASE: Emergenza
Emer: NOP   0;
      S     #ModoEmergenza;
      R     #ModoTestMacchina;
      R     #ModoSetup;
      R     #ModoManuale;
      R     #ModoAutomatico;
      JU    END;
NETWORK
TITLE = CASE: Test Ausiliari
Test: NOP   0;
      R     #ModoEmergenza;
      S     #ModoTestMacchina;
      R     #ModoSetup;
      R     #ModoManuale;
      R     #ModoAutomatico;
      JU    END;
NETWORK
TITLE = CASE: Modo setup
Setu: NOP   0;
      R     #ModoEmergenza;
      R     #ModoTestMacchina;
      S     #ModoSetup;
      R     #ModoManuale;
      R     #ModoAutomatico;
      JU    END;
NETWORK
TITLE = CASE: Modo Manuale
Manu: NOP   0;
      R     #ModoEmergenza;
      R     #ModoTestMacchina;
      R     #ModoSetup;
      S     #ModoManuale;
      R     #ModoAutomatico;
      JU    END;
NETWORK
TITLE = CASE: Modo Automatico
Auto: NOP   0;
      R     #ModoEmergenza;
      R     #ModoTestMacchina;
      R     #ModoSetup;
      R     #ModoManuale;
      S     #ModoAutomatico;
      JU    END;
NETWORK
TITLE = END CASE
END:  NOP   0;
NETWORK
TITLE = Usita Digitale PlcOk
      AN    #AllarmeEmergenza;
      =     #DO_PlcOk;
END_FUNCTION

FUNCTION "Bench.Alarms" : VOID	// FC 21
VERSION : 0.1
VAR_INPUT
  NumDBallarmi : BLOCK_DB ;
  Reset_Allarmi : BOOL ;
END_VAR
VAR_OUTPUT
  AllarmeEmergenza : BOOL ;
  AllarmeStopCiclo : BOOL ;
  AllarmeStartCiclo : BOOL ;
  AllarmeWarning : BOOL ;
END_VAR
VAR_TEMP
  Appoggio : ARRAY  [1 .. 8 ] OF BOOL ;
  Index : INT ;
END_VAR
BEGIN
NETWORK
TITLE = Allarmi Emergenza: Byte 0:7
      OPN   #NumDBallarmi;
      L     DBD 0;
      L     0;
      ==D;
      =     #Appoggio[1];
      L     DBD 4;
      L     0;
      ==D;
      =     #Appoggio[2];
      A     #Appoggio[1];
      A     #Appoggio[2];
      NOT;
      =     #AllarmeEmergenza;
NETWORK
TITLE = Allarmi StopCiclo: Byte 8:15
      L     DBD 8;
      L     0;
      ==D;
      =     #Appoggio[3];
      L     DBD 12;
      L     0;
      ==D;
      =     #Appoggio[4];
      A     #Appoggio[3];
      A     #Appoggio[4];
      NOT;
      O     #AllarmeEmergenza;
      =     #AllarmeStopCiclo;
NETWORK
TITLE = Allarmi StarCiclo: Byte 16:23
      L     DBD 16;
      L     0;
      ==D;
      =     #Appoggio[5];
      L     DBD 20;
      L     0;
      ==D;
      =     #Appoggio[6];
      A     #Appoggio[5];
      A     #Appoggio[6];
      NOT;
      O     #AllarmeEmergenza;
      =     #AllarmeStartCiclo;
NETWORK
TITLE = Allarmi Warning: Byte 24:30
      L     DBD 24;
      L     0;
      ==D;
      =     #Appoggio[7];
      L     DBD 28;
      L     0;
      ==D;
      =     #Appoggio[8];
      A     #Appoggio[7];
      A     #Appoggio[8];
      NOT;
      =     #AllarmeWarning;
NETWORK
TITLE = Reset di tutti gli Allarmi
      A     #Reset_Allarmi;
      JCN   end;
      L     8;
Znxt: T     #Index;
      L     1;
      -D;
      SLD   5;	//Colcolo l'indirizzo della DBD (#Index * 8 * 4)
      LAR1;
      L     0;
      T     DBD [AR1,P#0.0];
      L     #Index;
      LOOP  Znxt;
end:  NOP   0;
END_FUNCTION

// FC 40: know-how protected block, not included

